LIN {X 0,Y 409.933,Z 400.183,A -85,B 0,C 180,E1 -10526.068,E2 -10526.068} C_VEL
LIN {X 0,Y 409.928,Z 401.653,A -85,B 0,C 180,E1 -10527.052,E2 -10527.052} C_VEL
LIN {X 0,Y 409.968,Z 402.683,A -85,B 0,C 180,E1 -10528.035,E2 -10528.035} C_VEL
LIN {X 0,Y 409.937,Z 403.318,A -85,B 0,C 180,E1 -10529.018,E2 -10529.018} C_VEL
LIN {X 0,Y 409.927,Z 403.562,A -85,B 0,C 180,E1 -10530,E2 -10530} C_VEL
LIN {X 0,Y 409.937,Z 403.388,A -85,B 0,C 180,E1 -10530.982,E2 -10530.982} C_VEL
LIN {X 0,Y 409.968,Z 402.792,A -85,B 0,C 180,E1 -10531.965,E2 -10531.965} C_VEL
LIN {X 0,Y 409.933,Z 400.415,A -85,B 0,C 180,E1 -10533.932,E2 -10533.932} C_VEL
LIN {X 0,Y 410.02,Z 397.492,A -85,B 0,C 180,E1 -10535.409,E2 -10535.409} C_VEL
LIN {X 0,Y 410.169,Z 393.533,A -85,B 0,C 180,E1 -10536.888,E2 -10536.888} C_VEL
LIN {X 0,Y 410.424,Z 388.44,A -85,B 0,C 180,E1 -10538.369,E2 -10538.369} C_VEL
LIN {X 0,Y 410.834,Z 382.051,A -85,B 0,C 180,E1 -10539.849,E2 -10539.849} C_VEL
LIN {X 0,Y 411.43,Z 374.069,A -85,B 0,C 180,E1 -10541.329,E2 -10541.329} C_VEL
LIN {X 0,Y 412.303,Z 364.173,A -85,B 0,C 180,E1 -10542.802,E2 -10542.802} C_VEL
LIN {X 0,Y 412.887,Z 354.848,A -85,B 0,C 180,E1 -10543.93,E2 -10543.93} C_VEL
LIN {X 0,Y 413.712,Z 343.698,A -85,B 0,C 180,E1 -10545.014,E2 -10545.014} C_VEL
LIN {X 0,Y 414.567,Z 332.678,A -85,B 0,C 180,E1 -10545.864,E2 -10545.864} C_VEL
LIN {X 0,Y 414.903,Z 324.983,A -85,B 0,C 180,E1 -10546.356,E2 -10546.356} C_VEL
LIN {X 0,Y 413.288,Z 311.721,A -85,B 0,C 180,E1 -10547.105,E2 -10547.105} C_VEL
LIN {X 0,Y 410.881,Z 298.907,A -85,B 0,C 180,E1 -10547.674,E2 -10547.674} C_VEL
LIN {X 0,Y 410.406,Z 296.498,A -85,B 0,C 180,E1 -10547.759,E2 -10547.759} C_VEL
LIN {X 0,Y 410.712,Z 289.615,A -85,B 0,C 180,E1 -10551.059,E2 -10551.059} C_VEL
LIN {X 0,Y 410.994,Z 283.191,A -85,B 0,C 180,E1 -10554.229,E2 -10554.229} C_VEL
LIN {X 0,Y 411.373,Z 276.838,A -85,B 0,C 180,E1 -10557.469,E2 -10557.469} C_VEL
LIN {X 0,Y 411.844,Z 270.571,A -85,B 0,C 180,E1 -10560.792,E2 -10560.792} C_VEL
LIN {X 0,Y 412.452,Z 264.434,A -85,B 0,C 180,E1 -10564.214,E2 -10564.214} C_VEL
LIN {X 0,Y 412.379,Z 260.162,A -85,B 0,C 180,E1 -10566.773,E2 -10566.773} C_VEL
LIN {X 0,Y 411.758,Z 255.497,A -85,B 0,C 180,E1 -10569.818,E2 -10569.818} C_VEL
LIN {X 0,Y 411.207,Z 252.267,A -85,B 0,C 180,E1 -10572.13,E2 -10572.13} C_VEL
LIN {X 0,Y 411.176,Z 252.27,A -85,B 0,C 180,E1 -10575.509,E2 -10575.509} C_VEL
LIN {X 0,Y 411.199,Z 252.27,A -85,B 0,C 180,E1 -10578.765,E2 -10578.765} C_VEL
LIN {X 0,Y 411.203,Z 252.267,A -85,B 0,C 180,E1 -10582.026,E2 -10582.026} C_VEL
LIN {X 0,Y 411.204,Z 252.266,A -85,B 0,C 180,E1 -10585.665,E2 -10585.665} C_VEL
LIN {X 0,Y 411.195,Z 252.267,A -85,B 0,C 180,E1 -10589.152,E2 -10589.152} C_VEL
LIN {X 0,Y 411.256,Z 252.258,A -85,B 0,C 180,E1 -10592.521,E2 -10592.521} C_VEL
LIN {X 0,Y 411.223,Z 252.264,A -85,B 0,C 180,E1 -10595.783,E2 -10595.783} C_VEL
LIN {X 0,Y 411.191,Z 252.267,A -85,B 0,C 180,E1 -10598.965,E2 -10598.965} C_VEL
LIN {X 0,Y 411.247,Z 252.262,A -85,B 0,C 180,E1 -10602.084,E2 -10602.084} C_VEL
LIN {X 0,Y 411.254,Z 252.26,A -85,B 0,C 180,E1 -10605.146,E2 -10605.146} C_VEL
LIN {X 0,Y 411.279,Z 252.257,A -85,B 0,C 180,E1 -10608.166,E2 -10608.166} C_VEL
LIN {X 0,Y 411.475,Z 252.232,A -85,B 0,C 180,E1 -10612.145,E2 -10612.145} C_VEL
LIN {X 0,Y 411.468,Z 252.233,A -85,B 0,C 180,E1 -10614.117,E2 -10614.117} C_VEL
LIN {X 0,Y 411.506,Z 252.228,A -85,B 0,C 180,E1 -10618.041,E2 -10618.041} C_VEL
LIN {X 0,Y 411.634,Z 252.212,A -85,B 0,C 180,E1 -10619.999,E2 -10619.999} C_VEL
LIN {X 0,Y 411.46,Z 252.236,A -85,B 0,C 180,E1 -10622.936,E2 -10622.936} C_VEL
LIN {X 0,Y 411.452,Z 252.236,A -85,B 0,C 180,E1 -10626.866,E2 -10626.866} C_VEL
LIN {X 0,Y 411.354,Z 252.446,A -85,B 0,C 180,E1 -10628.844,E2 -10628.844} C_VEL
LIN {X 0,Y 411.368,Z 255.81,A -85,B 0,C 180,E1 -10631.829,E2 -10631.829} C_VEL
LIN {X 0,Y 411.223,Z 258.159,A -85,B 0,C 180,E1 -10633.842,E2 -10633.842} C_VEL
LIN {X 0,Y 411.047,Z 261.892,A -85,B 0,C 180,E1 -10636.896,E2 -10636.896} C_VEL
LIN {X 0,Y 410.791,Z 265.812,A -85,B 0,C 180,E1 -10640.008,E2 -10640.008} C_VEL
LIN {X 0,Y 410.58,Z 269.911,A -85,B 0,C 180,E1 -10643.183,E2 -10643.183} C_VEL
LIN {X 0,Y 410.391,Z 274.236,A -85,B 0,C 180,E1 -10646.438,E2 -10646.438} C_VEL
LIN {X 0,Y 410.331,Z 276.757,A -85,B 0,C 180,E1 -10648.307,E2 -10648.307} C_VEL
LIN {X 0,Y 414.045,Z 291.96,A -85,B 0,C 180,E1 -10649.053,E2 -10649.053} C_VEL
LIN {X 0,Y 415.423,Z 299.541,A -85,B 0,C 180,E1 -10649.501,E2 -10649.501} C_VEL
LIN {X 0,Y 414.931,Z 311.573,A -85,B 0,C 180,E1 -10650.253,E2 -10650.253} C_VEL
LIN {X 0,Y 414.2,Z 322.984,A -85,B 0,C 180,E1 -10651.164,E2 -10651.164} C_VEL
LIN {X 0,Y 413.404,Z 333.611,A -85,B 0,C 180,E1 -10652.232,E2 -10652.232} C_VEL
LIN {X 0,Y 412.54,Z 344.203,A -85,B 0,C 180,E1 -10653.568,E2 -10653.568} C_VEL
LIN {X 0,Y 411.775,Z 353.273,A -85,B 0,C 180,E1 -10654.993,E2 -10654.993} C_VEL
LIN {X 0,Y 411.141,Z 361.113,A -85,B 0,C 180,E1 -10656.545,E2 -10656.545} C_VEL
LIN {X 0,Y 410.667,Z 367.275,A -85,B 0,C 180,E1 -10658.075,E2 -10658.075} C_VEL
LIN {X 0,Y 410.326,Z 372.035,A -85,B 0,C 180,E1 -10659.58,E2 -10659.58} C_VEL
LIN {X 0,Y 410.099,Z 375.597,A -85,B 0,C 180,E1 -10661.06,E2 -10661.06} C_VEL
LIN {X 0,Y 409.93,Z 378.103,A -85,B 0,C 180,E1 -10662.507,E2 -10662.507} C_VEL
LIN {X 0,Y 409.84,Z 379.686,A -85,B 0,C 180,E1 -10663.929,E2 -10663.929} C_VEL
LIN {X 0,Y 409.775,Z 380.432,A -85,B 0,C 180,E1 -10665.318,E2 -10665.318} C_VEL
LIN {X 0,Y 409.739,Z 380.392,A -85,B 0,C 180,E1 -10666.679,E2 -10666.679} C_VEL
LIN {X 0,Y 409.781,Z 379.571,A -85,B 0,C 180,E1 -10668.021,E2 -10668.021} C_VEL
LIN {X 0,Y 409.877,Z 378.049,A -85,B 0,C 180,E1 -10669.341,E2 -10669.341} C_VEL
LIN {X 0,Y 410.003,Z 375.839,A -85,B 0,C 180,E1 -10670.638,E2 -10670.638} C_VEL
LIN {X 0,Y 410.322,Z 370.969,A -85,B 0,C 180,E1 -10672.595,E2 -10672.595} C_VEL
LIN {X 0,Y 410.649,Z 366.267,A -85,B 0,C 180,E1 -10674.002,E2 -10674.002} C_VEL
LIN {X 0,Y 411.05,Z 359.297,A -85,B 0,C 180,E1 -10675.653,E2 -10675.653} C_VEL
LIN {X 0,Y 411.696,Z 351.038,A -85,B 0,C 180,E1 -10677.181,E2 -10677.181} C_VEL
LIN {X 0,Y 412.311,Z 342.559,A -85,B 0,C 180,E1 -10678.456,E2 -10678.456} C_VEL
LIN {X 0,Y 412.941,Z 333,A -85,B 0,C 180,E1 -10679.636,E2 -10679.636} C_VEL
LIN {X 0,Y 413.603,Z 323.215,A -85,B 0,C 180,E1 -10680.618,E2 -10680.618} C_VEL
LIN {X 0,Y 414.317,Z 311.202,A -85,B 0,C 180,E1 -10681.575,E2 -10681.575} C_VEL
LIN {X 0,Y 414.99,Z 300.07,A -85,B 0,C 180,E1 -10682.261,E2 -10682.261} C_VEL
LIN {X 0,Y 412.651,Z 287.184,A -85,B 0,C 180,E1 -10682.965,E2 -10682.965} C_VEL
LIN {X 0,Y 410.191,Z 276.058,A -85,B 0,C 180,E1 -10683.425,E2 -10683.425} C_VEL
LIN {X 0,Y 410.335,Z 271.318,A -85,B 0,C 180,E1 -10686.801,E2 -10686.801} C_VEL
LIN {X 0,Y 410.554,Z 266.488,A -85,B 0,C 180,E1 -10690.302,E2 -10690.302} C_VEL
LIN {X 0,Y 410.726,Z 262.34,A -85,B 0,C 180,E1 -10693.374,E2 -10693.374} C_VEL
LIN {X 0,Y 410.976,Z 257.338,A -85,B 0,C 180,E1 -10697.156,E2 -10697.156} C_VEL
LIN {X 0,Y 411.091,Z 253.482,A -85,B 0,C 180,E1 -10700.157,E2 -10700.157} C_VEL
LIN {X 0,Y 411.12,Z 252.276,A -85,B 0,C 180,E1 -10701.15,E2 -10701.15} C_VEL
LIN {X 0,Y 411.404,Z 252.241,A -85,B 0,C 180,E1 -10703.132,E2 -10703.132} C_VEL
LIN {X 0,Y 411.301,Z 252.252,A -85,B 0,C 180,E1 -10705.099,E2 -10705.099} C_VEL
LIN {X 0,Y 411.481,Z 252.228,A -85,B 0,C 180,E1 -10708.307,E2 -10708.307} C_VEL
LIN {X 0,Y 411.633,Z 252.211,A -85,B 0,C 180,E1 -10710,E2 -10710} C_VEL
LIN {X 0,Y 411.46,Z 252.231,A -85,B 0,C 180,E1 -10712.571,E2 -10712.571} C_VEL
LIN {X 0,Y 410.775,Z 252.318,A -85,B 0,C 180,E1 -10713.387,E2 -10713.387} C_VEL
LIN {X 0,Y 407.897,Z 252.677,A -85,B 0,C 180,E1 -10714.712,E2 -10714.712} C_VEL
LIN {X 0,Y 405.484,Z 252.976,A -85,B 0,C 180,E1 -10715.783,E2 -10715.783} C_VEL
LIN {X 0,Y 404.469,Z 253.105,A -85,B 0,C 180,E1 -10716.611,E2 -10716.611} C_VEL
LIN {X 0,Y 404.397,Z 253.11,A -85,B 0,C 180,E1 -10716.891,E2 -10716.891} C_VEL
LIN {X 0,Y 404.286,Z 253.125,A -85,B 0,C 180,E1 -10719.001,E2 -10719.001} C_VEL
LIN {X 0,Y 404.26,Z 253.131,A -85,B 0,C 180,E1 -10722.041,E2 -10722.041} C_VEL
LIN {X 0,Y 404.202,Z 253.135,A -85,B 0,C 180,E1 -10725.118,E2 -10725.118} C_VEL
LIN {X 0,Y 404.203,Z 253.138,A -85,B 0,C 180,E1 -10728.238,E2 -10728.238} C_VEL
LIN {X 0,Y 404.169,Z 253.14,A -85,B 0,C 180,E1 -10731.417,E2 -10731.417} C_VEL
LIN {X 0,Y 404.167,Z 253.14,A -85,B 0,C 180,E1 -10734.666,E2 -10734.666} C_VEL
LIN {X 0,Y 404.187,Z 253.14,A -85,B 0,C 180,E1 -10738,E2 -10738} C_VEL
LIN {X 0,Y 404.135,Z 253.146,A -85,B 0,C 180,E1 -10741.56,E2 -10741.56} C_VEL
LIN {X 0,Y 404.174,Z 253.139,A -85,B 0,C 180,E1 -10745.017,E2 -10745.017} C_VEL
LIN {X 0,Y 404.153,Z 253.14,A -85,B 0,C 180,E1 -10748.756,E2 -10748.756} C_VEL
LIN {X 0,Y 404.181,Z 253.141,A -85,B 0,C 180,E1 -10751.611,E2 -10751.611} C_VEL
LIN {X 0,Y 404.19,Z 253.136,A -85,B 0,C 180,E1 -10754.531,E2 -10754.531} C_VEL
LIN {X 0,Y 404.196,Z 253.139,A -85,B 0,C 180,E1 -10757.306,E2 -10757.306} C_VEL
LIN {X 0,Y 404.158,Z 253.141,A -85,B 0,C 180,E1 -10759.956,E2 -10759.956} C_VEL
LIN {X 0,Y 404.131,Z 253.147,A -85,B 0,C 180,E1 -10763.125,E2 -10763.125} C_VEL
LIN {X 0,Y 404.135,Z 253.143,A -85,B 0,C 180,E1 -10766.189,E2 -10766.189} C_VEL
LIN {X 0,Y 404.144,Z 253.142,A -85,B 0,C 180,E1 -10769.716,E2 -10769.716} C_VEL
LIN {X 0,Y 404.186,Z 253.14,A -85,B 0,C 180,E1 -10773.124,E2 -10773.124} C_VEL
LIN {X 0,Y 404.168,Z 253.141,A -85,B 0,C 180,E1 -10775.335,E2 -10775.335} C_VEL
LIN {X 0,Y 404.13,Z 253.147,A -85,B 0,C 180,E1 -10778.582,E2 -10778.582} C_VEL
LIN {X 0,Y 404.202,Z 253.135,A -85,B 0,C 180,E1 -10781.763,E2 -10781.763} C_VEL
LIN {X 0,Y 404.198,Z 253.139,A -85,B 0,C 180,E1 -10784.883,E2 -10784.883} C_VEL
LIN {X 0,Y 404.249,Z 253.13,A -85,B 0,C 180,E1 -10787.96,E2 -10787.96} C_VEL
LIN {X 0,Y 404.398,Z 253.113,A -85,B 0,C 180,E1 -10792.13,E2 -10792.13} C_VEL
LIN {X 0,Y 404.416,Z 253.111,A -85,B 0,C 180,E1 -10794.016,E2 -10794.016} C_VEL
LIN {X 0,Y 404.476,Z 253.103,A -85,B 0,C 180,E1 -10798.01,E2 -10798.01} C_VEL
LIN {X 0,Y 404.605,Z 253.088,A -85,B 0,C 180,E1 -10800.001,E2 -10800.001} C_VEL
LIN {X 0,Y 404.418,Z 253.108,A -85,B 0,C 180,E1 -10802.99,E2 -10802.99} C_VEL
LIN {X 0,Y 404.406,Z 253.109,A -85,B 0,C 180,E1 -10806.988,E2 -10806.988} C_VEL
LIN {X 0,Y 404.266,Z 253.13,A -85,B 0,C 180,E1 -10810.013,E2 -10810.013} C_VEL
LIN {X 0,Y 404.263,Z 253.128,A -85,B 0,C 180,E1 -10813.213,E2 -10813.213} C_VEL
LIN {X 0,Y 404.212,Z 253.133,A -85,B 0,C 180,E1 -10817.008,E2 -10817.008} C_VEL
LIN {X 0,Y 404.161,Z 253.14,A -85,B 0,C 180,E1 -10820.353,E2 -10820.353} C_VEL
LIN {X 0,Y 404.167,Z 253.143,A -85,B 0,C 180,E1 -10823.576,E2 -10823.576} C_VEL
LIN {X 0,Y 404.182,Z 253.141,A -85,B 0,C 180,E1 -10825.768,E2 -10825.768} C_VEL
LIN {X 0,Y 404.193,Z 253.138,A -85,B 0,C 180,E1 -10828.001,E2 -10828.001} C_VEL
LIN {X 0,Y 404.138,Z 253.146,A -85,B 0,C 180,E1 -10831.559,E2 -10831.559} C_VEL
LIN {X 0,Y 404.184,Z 253.14,A -85,B 0,C 180,E1 -10835.017,E2 -10835.017} C_VEL
LIN {X 0,Y 404.157,Z 253.142,A -85,B 0,C 180,E1 -10838.758,E2 -10838.758} C_VEL
LIN {X 0,Y 404.123,Z 253.146,A -85,B 0,C 180,E1 -10841.601,E2 -10841.601} C_VEL
LIN {X 0,Y 404.146,Z 253.143,A -85,B 0,C 180,E1 -10844.523,E2 -10844.523} C_VEL
LIN {X 0,Y 404.137,Z 253.147,A -85,B 0,C 180,E1 -10847.297,E2 -10847.297} C_VEL
LIN {X 0,Y 404.193,Z 253.241,A -85,B 0,C 180,E1 -10849.222,E2 -10849.222} C_VEL
LIN {X 0,Y 405.002,Z 257.819,A -85,B 0,C 180,E1 -10852.003,E2 -10852.003} C_VEL
LIN {X 0,Y 405.39,Z 262.275,A -85,B 0,C 180,E1 -10854.57,E2 -10854.57} C_VEL
LIN {X 0,Y 405.055,Z 267.592,A -85,B 0,C 180,E1 -10857.462,E2 -10857.462} C_VEL
LIN {X 0,Y 404.493,Z 274.108,A -85,B 0,C 180,E1 -10860.89,E2 -10860.89} C_VEL
LIN {X 0,Y 404.056,Z 281.663,A -85,B 0,C 180,E1 -10864.753,E2 -10864.753} C_VEL
LIN {X 0,Y 403.719,Z 288.235,A -85,B 0,C 180,E1 -10868.021,E2 -10868.021} C_VEL
LIN {X 0,Y 403.451,Z 294.748,A -85,B 0,C 180,E1 -10871.2,E2 -10871.2} C_VEL
LIN {X 0,Y 403.357,Z 297.222,A -85,B 0,C 180,E1 -10872.308,E2 -10872.308} C_VEL
LIN {X 0,Y 405.673,Z 310.351,A -85,B 0,C 180,E1 -10872.827,E2 -10872.827} C_VEL
LIN {X 0,Y 407.456,Z 323.993,A -85,B 0,C 180,E1 -10873.57,E2 -10873.57} C_VEL
LIN {X 0,Y 407.412,Z 330.524,A -85,B 0,C 180,E1 -10873.978,E2 -10873.978} C_VEL
LIN {X 0,Y 406.585,Z 342.104,A -85,B 0,C 180,E1 -10874.844,E2 -10874.844} C_VEL
LIN {X 0,Y 405.723,Z 353.789,A -85,B 0,C 180,E1 -10875.965,E2 -10875.965} C_VEL
LIN {X 0,Y 405.064,Z 364.197,A -85,B 0,C 180,E1 -10877.22,E2 -10877.22} C_VEL
LIN {X 0,Y 404.208,Z 374.12,A -85,B 0,C 180,E1 -10878.72,E2 -10878.72} C_VEL
LIN {X 0,Y 403.675,Z 382.113,A -85,B 0,C 180,E1 -10880.227,E2 -10880.227} C_VEL
LIN {X 0,Y 403.366,Z 387.519,A -85,B 0,C 180,E1 -10881.483,E2 -10881.483} C_VEL
LIN {X 0,Y 403.082,Z 392.807,A -85,B 0,C 180,E1 -10882.99,E2 -10882.99} C_VEL
LIN {X 0,Y 402.918,Z 396.908,A -85,B 0,C 180,E1 -10884.495,E2 -10884.495} C_VEL
LIN {X 0,Y 402.854,Z 399.941,A -85,B 0,C 180,E1 -10885.998,E2 -10885.998} C_VEL
LIN {X 0,Y 402.827,Z 401.426,A -85,B 0,C 180,E1 -10887,E2 -10887} C_VEL
LIN {X 0,Y 402.866,Z 402.464,A -85,B 0,C 180,E1 -10888,E2 -10888} C_VEL
LIN {X 0,Y 402.864,Z 403.106,A -85,B 0,C 180,E1 -10889,E2 -10889} C_VEL
LIN {X 0,Y 402.852,Z 403.358,A -85,B 0,C 180,E1 -10890,E2 -10890} C_VEL
LIN {X 0,Y 402.864,Z 403.199,A -85,B 0,C 180,E1 -10890.999,E2 -10890.999} C_VEL
LIN {X 0,Y 402.866,Z 402.609,A -85,B 0,C 180,E1 -10891.999,E2 -10891.999} C_VEL
LIN {X 0,Y 402.853,Z 400.245,A -85,B 0,C 180,E1 -10894.001,E2 -10894.001} C_VEL
LIN {X 0,Y 402.918,Z 397.334,A -85,B 0,C 180,E1 -10895.505,E2 -10895.505} C_VEL
LIN {X 0,Y 403.082,Z 393.389,A -85,B 0,C 180,E1 -10897.01,E2 -10897.01} C_VEL
LIN {X 0,Y 403.366,Z 388.31,A -85,B 0,C 180,E1 -10898.516,E2 -10898.516} C_VEL
LIN {X 0,Y 403.824,Z 381.942,A -85,B 0,C 180,E1 -10900.022,E2 -10900.022} C_VEL
LIN {X 0,Y 404.429,Z 373.983,A -85,B 0,C 180,E1 -10901.527,E2 -10901.527} C_VEL
LIN {X 0,Y 405.353,Z 364.109,A -85,B 0,C 180,E1 -10903.026,E2 -10903.026} C_VEL
LIN {X 0,Y 406.022,Z 354.346,A -85,B 0,C 180,E1 -10904.225,E2 -10904.225} C_VEL
LIN {X 0,Y 406.861,Z 343.762,A -85,B 0,C 180,E1 -10905.273,E2 -10905.273} C_VEL
LIN {X 0,Y 407.75,Z 332.866,A -85,B 0,C 180,E1 -10906.134,E2 -10906.134} C_VEL
LIN {X 0,Y 408.015,Z 325.458,A -85,B 0,C 180,E1 -10906.628,E2 -10906.628} C_VEL
LIN {X 0,Y 406.532,Z 312.758,A -85,B 0,C 180,E1 -10907.375,E2 -10907.375} C_VEL
LIN {X 0,Y 404.064,Z 299.804,A -85,B 0,C 180,E1 -10907.982,E2 -10907.982} C_VEL
LIN {X 0,Y 403.377,Z 296.306,A -85,B 0,C 180,E1 -10908.112,E2 -10908.112} C_VEL
LIN {X 0,Y 403.662,Z 289.507,A -85,B 0,C 180,E1 -10911.445,E2 -10911.445} C_VEL
LIN {X 0,Y 404.001,Z 283.107,A -85,B 0,C 180,E1 -10914.676,E2 -10914.676} C_VEL
LIN {X 0,Y 404.388,Z 276.776,A -85,B 0,C 180,E1 -10917.984,E2 -10917.984} C_VEL
LIN {X 0,Y 405.008,Z 269.916,A -85,B 0,C 180,E1 -10921.756,E2 -10921.756} C_VEL
LIN {X 0,Y 405.468,Z 264.438,A -85,B 0,C 180,E1 -10924.888,E2 -10924.888} C_VEL
LIN {X 0,Y 405.286,Z 260.478,A -85,B 0,C 180,E1 -10927.367,E2 -10927.367} C_VEL
LIN {X 0,Y 404.687,Z 256.34,A -85,B 0,C 180,E1 -10930.17,E2 -10930.17} C_VEL
LIN {X 0,Y 404.159,Z 253.144,A -85,B 0,C 180,E1 -10932.557,E2 -10932.557} C_VEL
LIN {X 0,Y 404.148,Z 253.147,A -85,B 0,C 180,E1 -10935.925,E2 -10935.925} C_VEL
LIN {X 0,Y 404.151,Z 253.147,A -85,B 0,C 180,E1 -10938.638,E2 -10938.638} C_VEL
LIN {X 0,Y 404.16,Z 253.145,A -85,B 0,C 180,E1 -10941.489,E2 -10941.489} C_VEL
LIN {X 0,Y 404.183,Z 253.14,A -85,B 0,C 180,E1 -10944.983,E2 -10944.983} C_VEL
LIN {X 0,Y 404.143,Z 253.145,A -85,B 0,C 180,E1 -10948.553,E2 -10948.553} C_VEL
LIN {X 0,Y 404.194,Z 253.138,A -85,B 0,C 180,E1 -10951.999,E2 -10951.999} C_VEL
LIN {X 0,Y 404.173,Z 253.141,A -85,B 0,C 180,E1 -10955.333,E2 -10955.333} C_VEL
LIN {X 0,Y 404.134,Z 253.146,A -85,B 0,C 180,E1 -10958.579,E2 -10958.579} C_VEL
LIN {X 0,Y 404.205,Z 253.137,A -85,B 0,C 180,E1 -10961.761,E2 -10961.761} C_VEL
LIN {X 0,Y 404.2,Z 253.138,A -85,B 0,C 180,E1 -10964.881,E2 -10964.881} C_VEL
LIN {X 0,Y 404.251,Z 253.131,A -85,B 0,C 180,E1 -10967.957,E2 -10967.957} C_VEL
LIN {X 0,Y 404.427,Z 253.11,A -85,B 0,C 180,E1 -10972.098,E2 -10972.098} C_VEL
LIN {X 0,Y 404.417,Z 253.111,A -85,B 0,C 180,E1 -10974.014,E2 -10974.014} C_VEL
LIN {X 0,Y 404.475,Z 253.104,A -85,B 0,C 180,E1 -10978.007,E2 -10978.007} C_VEL
LIN {X 0,Y 404.603,Z 253.088,A -85,B 0,C 180,E1 -10979.999,E2 -10979.999} C_VEL
LIN {X 0,Y 404.417,Z 253.114,A -85,B 0,C 180,E1 -10982.987,E2 -10982.987} C_VEL
LIN {X 0,Y 404.398,Z 253.115,A -85,B 0,C 180,E1 -10986.986,E2 -10986.986} C_VEL
LIN {X 0,Y 404.376,Z 253.118,A -85,B 0,C 180,E1 -10987.991,E2 -10987.991} C_VEL
LIN {X 0,Y 404.365,Z 253.737,A -85,B 0,C 180,E1 -10988.998,E2 -10988.998} C_VEL
LIN {X 0,Y 404.334,Z 257.099,A -85,B 0,C 180,E1 -10992.038,E2 -10992.038} C_VEL
LIN {X 0,Y 404.097,Z 260.696,A -85,B 0,C 180,E1 -10995.121,E2 -10995.121} C_VEL
LIN {X 0,Y 403.875,Z 264.511,A -85,B 0,C 180,E1 -10998.252,E2 -10998.252} C_VEL
LIN {X 0,Y 403.632,Z 268.511,A -85,B 0,C 180,E1 -11001.446,E2 -11001.446} C_VEL
LIN {X 0,Y 403.429,Z 273.172,A -85,B 0,C 180,E1 -11005.062,E2 -11005.062} C_VEL
LIN {X 0,Y 403.272,Z 276.979,A -85,B 0,C 180,E1 -11007.947,E2 -11007.947} C_VEL
LIN {X 0,Y 406.97,Z 291.921,A -85,B 0,C 180,E1 -11008.703,E2 -11008.703} C_VEL
LIN {X 0,Y 408.755,Z 302.254,A -85,B 0,C 180,E1 -11009.34,E2 -11009.34} C_VEL
LIN {X 0,Y 408.087,Z 313.529,A -85,B 0,C 180,E1 -11010.081,E2 -11010.081} C_VEL
LIN {X 0,Y 407.324,Z 324.098,A -85,B 0,C 180,E1 -11010.963,E2 -11010.963} C_VEL
LIN {X 0,Y 406.464,Z 334.838,A -85,B 0,C 180,E1 -11012.089,E2 -11012.089} C_VEL
LIN {X 0,Y 405.606,Z 344.714,A -85,B 0,C 180,E1 -11013.372,E2 -11013.372} C_VEL
LIN {X 0,Y 404.89,Z 352.697,A -85,B 0,C 180,E1 -11014.642,E2 -11014.642} C_VEL
LIN {X 0,Y 404.27,Z 359.623,A -85,B 0,C 180,E1 -11015.978,E2 -11015.978} C_VEL
LIN {X 0,Y 403.743,Z 366.123,A -85,B 0,C 180,E1 -11017.533,E2 -11017.533} C_VEL
LIN {X 0,Y 403.29,Z 372.051,A -85,B 0,C 180,E1 -11019.377,E2 -11019.377} C_VEL
LIN {X 0,Y 403.047,Z 375.464,A -85,B 0,C 180,E1 -11020.788,E2 -11020.788} C_VEL
LIN {X 0,Y 402.862,Z 377.979,A -85,B 0,C 180,E1 -11022.192,E2 -11022.192} C_VEL
LIN {X 0,Y 402.824,Z 378.914,A -85,B 0,C 180,E1 -11022.883,E2 -11022.883} C_VEL
LIN {X 0,Y 402.731,Z 380.235,A -85,B 0,C 180,E1 -11024.318,E2 -11024.318} C_VEL
LIN {X 0,Y 402.678,Z 380.697,A -85,B 0,C 180,E1 -11025.725,E2 -11025.725} C_VEL
LIN {X 0,Y 402.65,Z 380.375,A -85,B 0,C 180,E1 -11027.143,E2 -11027.143} C_VEL
LIN {X 0,Y 402.732,Z 379.19,A -85,B 0,C 180,E1 -11028.621,E2 -11028.621} C_VEL
LIN {X 0,Y 402.833,Z 377.042,A -85,B 0,C 180,E1 -11030.14,E2 -11030.14} C_VEL
LIN {X 0,Y 403.081,Z 373.838,A -85,B 0,C 180,E1 -11031.682,E2 -11031.682} C_VEL
LIN {X 0,Y 403.383,Z 369.38,A -85,B 0,C 180,E1 -11033.265,E2 -11033.265} C_VEL
LIN {X 0,Y 403.786,Z 363.222,A -85,B 0,C 180,E1 -11034.945,E2 -11034.945} C_VEL
LIN {X 0,Y 404.342,Z 355.751,A -85,B 0,C 180,E1 -11036.54,E2 -11036.54} C_VEL
LIN {X 0,Y 405.05,Z 346.647,A -85,B 0,C 180,E1 -11038.08,E2 -11038.08} C_VEL
LIN {X 0,Y 405.736,Z 336.849,A -85,B 0,C 180,E1 -11039.415,E2 -11039.415} C_VEL
LIN {X 0,Y 406.522,Z 325.674,A -85,B 0,C 180,E1 -11040.624,E2 -11040.624} C_VEL
LIN {X 0,Y 407.287,Z 313.794,A -85,B 0,C 180,E1 -11041.643,E2 -11041.643} C_VEL
LIN {X 0,Y 407.973,Z 302.84,A -85,B 0,C 180,E1 -11042.37,E2 -11042.37} C_VEL
LIN {X 0,Y 407.917,Z 299.95,A -85,B 0,C 180,E1 -11042.539,E2 -11042.539} C_VEL
LIN {X 0,Y 405.529,Z 287.07,A -85,B 0,C 180,E1 -11043.254,E2 -11043.254} C_VEL
LIN {X 0,Y 403.138,Z 276.246,A -85,B 0,C 180,E1 -11043.711,E2 -11043.711} C_VEL
LIN {X 0,Y 403.223,Z 272.558,A -85,B 0,C 180,E1 -11046.367,E2 -11046.367} C_VEL
LIN {X 0,Y 403.455,Z 268.129,A -85,B 0,C 180,E1 -11049.612,E2 -11049.612} C_VEL
LIN {X 0,Y 403.659,Z 263.268,A -85,B 0,C 180,E1 -11053.248,E2 -11053.248} C_VEL
LIN {X 0,Y 403.894,Z 258.357,A -85,B 0,C 180,E1 -11057.009,E2 -11057.009} C_VEL
LIN {X 0,Y 404.034,Z 254.575,A -85,B 0,C 180,E1 -11059.983,E2 -11059.983} C_VEL
LIN {X 0,Y 404.074,Z 253.314,A -85,B 0,C 180,E1 -11060.994,E2 -11060.994} C_VEL
LIN {X 0,Y 404.341,Z 253.12,A -85,B 0,C 180,E1 -11063.012,E2 -11063.012} C_VEL
LIN {X 0,Y 404.272,Z 253.128,A -85,B 0,C 180,E1 -11065.014,E2 -11065.014} C_VEL
LIN {X 0,Y 404.473,Z 253.102,A -85,B 0,C 180,E1 -11068.009,E2 -11068.009} C_VEL
LIN {X 0,Y 404.602,Z 253.087,A -85,B 0,C 180,E1 -11070,E2 -11070} C_VEL
LIN {X 0,Y 404.414,Z 253.11,A -85,B 0,C 180,E1 -11072.989,E2 -11072.989} C_VEL
LIN {X 0,Y 404.397,Z 253.11,A -85,B 0,C 180,E1 -11076.891,E2 -11076.891} C_VEL
LIN {X 0,Y 403.746,Z 253.194,A -85,B 0,C 180,E1 -11077.722,E2 -11077.722} C_VEL
LIN {X 0,Y 400.847,Z 253.557,A -85,B 0,C 180,E1 -11079.069,E2 -11079.069} C_VEL
LIN {X 0,Y 398.367,Z 253.865,A -85,B 0,C 180,E1 -11080.158,E2 -11080.158} C_VEL
LIN {X 0,Y 397.29,Z 253.996,A -85,B 0,C 180,E1 -11081.001,E2 -11081.001} C_VEL
LIN {X 0,Y 397.197,Z 254.007,A -85,B 0,C 180,E1 -11081.287,E2 -11081.287} C_VEL
LIN {X 0,Y 397.172,Z 254.014,A -85,B 0,C 180,E1 -11084.343,E2 -11084.343} C_VEL
LIN {X 0,Y 397.165,Z 254.012,A -85,B 0,C 180,E1 -11087.507,E2 -11087.507} C_VEL
LIN {X 0,Y 397.122,Z 254.017,A -85,B 0,C 180,E1 -11090.729,E2 -11090.729} C_VEL
LIN {X 0,Y 397.124,Z 254.02,A -85,B 0,C 180,E1 -11094.018,E2 -11094.018} C_VEL
LIN {X 0,Y 397.184,Z 254.011,A -85,B 0,C 180,E1 -11097.39,E2 -11097.39} C_VEL
LIN {X 0,Y 397.075,Z 254.023,A -85,B 0,C 180,E1 -11100.882,E2 -11100.882} C_VEL
LIN {X 0,Y 397.115,Z 254.018,A -85,B 0,C 180,E1 -11104.494,E2 -11104.494} C_VEL
LIN {X 0,Y 397.099,Z 254.019,A -85,B 0,C 180,E1 -11108.275,E2 -11108.275} C_VEL
LIN {X 0,Y 397.146,Z 254.015,A -85,B 0,C 180,E1 -11111.994,E2 -11111.994} C_VEL
LIN {X 0,Y 397.14,Z 254.017,A -85,B 0,C 180,E1 -11115.06,E2 -11115.06} C_VEL
LIN {X 0,Y 397.145,Z 254.014,A -85,B 0,C 180,E1 -11118.008,E2 -11118.008} C_VEL
LIN {X 0,Y 397.1,Z 254.021,A -85,B 0,C 180,E1 -11121.727,E2 -11121.727} C_VEL
LIN {X 0,Y 397.116,Z 254.02,A -85,B 0,C 180,E1 -11125.508,E2 -11125.508} C_VEL
LIN {X 0,Y 397.075,Z 254.026,A -85,B 0,C 180,E1 -11129.119,E2 -11129.119} C_VEL
LIN {X 0,Y 397.186,Z 254.012,A -85,B 0,C 180,E1 -11132.611,E2 -11132.611} C_VEL
LIN {X 0,Y 397.124,Z 254.016,A -85,B 0,C 180,E1 -11135.983,E2 -11135.983} C_VEL
LIN {X 0,Y 397.13,Z 254.015,A -85,B 0,C 180,E1 -11139.706,E2 -11139.706} C_VEL
LIN {X 0,Y 397.174,Z 254.014,A -85,B 0,C 180,E1 -11142.846,E2 -11142.846} C_VEL
LIN {X 0,Y 397.221,Z 254.008,A -85,B 0,C 180,E1 -11146.704,E2 -11146.704} C_VEL
LIN {X 0,Y 397.211,Z 254.005,A -85,B 0,C 180,E1 -11149.81,E2 -11149.81} C_VEL
LIN {X 0,Y 397.346,Z 253.991,A -85,B 0,C 180,E1 -11152.889,E2 -11152.889} C_VEL
LIN {X 0,Y 397.248,Z 254.002,A -85,B 0,C 180,E1 -11154.926,E2 -11154.926} C_VEL
LIN {X 0,Y 397.445,Z 253.979,A -85,B 0,C 180,E1 -11157.974,E2 -11157.974} C_VEL
LIN {X 0,Y 397.574,Z 253.964,A -85,B 0,C 180,E1 -11160.001,E2 -11160.001} C_VEL
LIN {X 0,Y 397.376,Z 253.985,A -85,B 0,C 180,E1 -11163.043,E2 -11163.043} C_VEL
LIN {X 0,Y 397.359,Z 253.987,A -85,B 0,C 180,E1 -11167.113,E2 -11167.113} C_VEL
LIN {X 0,Y 397.224,Z 254.008,A -85,B 0,C 180,E1 -11170.192,E2 -11170.192} C_VEL
LIN {X 0,Y 397.223,Z 254.005,A -85,B 0,C 180,E1 -11173.322,E2 -11173.322} C_VEL
LIN {X 0,Y 397.179,Z 254.01,A -85,B 0,C 180,E1 -11177.156,E2 -11177.156} C_VEL
LIN {X 0,Y 397.1,Z 254.019,A -85,B 0,C 180,E1 -11180.731,E2 -11180.731} C_VEL
LIN {X 0,Y 397.13,Z 254.018,A -85,B 0,C 180,E1 -11184.019,E2 -11184.019} C_VEL
LIN {X 0,Y 397.192,Z 254.012,A -85,B 0,C 180,E1 -11187.391,E2 -11187.391} C_VEL
LIN {X 0,Y 397.077,Z 254.023,A -85,B 0,C 180,E1 -11190.884,E2 -11190.884} C_VEL
LIN {X 0,Y 397.125,Z 254.016,A -85,B 0,C 180,E1 -11194.494,E2 -11194.494} C_VEL
LIN {X 0,Y 397.105,Z 254.019,A -85,B 0,C 180,E1 -11198.276,E2 -11198.276} C_VEL
LIN {X 0,Y 397.089,Z 254.024,A -85,B 0,C 180,E1 -11200.91,E2 -11200.91} C_VEL
LIN {X 0,Y 397.101,Z 254.021,A -85,B 0,C 180,E1 -11203.65,E2 -11203.65} C_VEL
LIN {X 0,Y 397.103,Z 254.023,A -85,B 0,C 180,E1 -11206.522,E2 -11206.522} C_VEL
LIN {X 0,Y 397.133,Z 254.122,A -85,B 0,C 180,E1 -11209.014,E2 -11209.014} C_VEL
LIN {X 0,Y 397.935,Z 258.663,A -85,B 0,C 180,E1 -11211.82,E2 -11211.82} C_VEL
LIN {X 0,Y 398.355,Z 263.028,A -85,B 0,C 180,E1 -11214.395,E2 -11214.395} C_VEL
LIN {X 0,Y 398.038,Z 268.469,A -85,B 0,C 180,E1 -11217.418,E2 -11217.418} C_VEL
LIN {X 0,Y 397.433,Z 274.993,A -85,B 0,C 180,E1 -11220.903,E2 -11220.903} C_VEL
LIN {X 0,Y 396.961,Z 282.583,A -85,B 0,C 180,E1 -11224.856,E2 -11224.856} C_VEL
LIN {X 0,Y 396.622,Z 289.091,A -85,B 0,C 180,E1 -11228.154,E2 -11228.154} C_VEL
LIN {X 0,Y 396.337,Z 295.59,A -85,B 0,C 180,E1 -11231.387,E2 -11231.387} C_VEL
LIN {X 0,Y 396.285,Z 296.809,A -85,B 0,C 180,E1 -11231.987,E2 -11231.987} C_VEL
LIN {X 0,Y 398.934,Z 312.219,A -85,B 0,C 180,E1 -11232.647,E2 -11232.647} C_VEL
LIN {X 0,Y 400.605,Z 325.587,A -85,B 0,C 180,E1 -11233.415,E2 -11233.415} C_VEL
LIN {X 0,Y 400.085,Z 336.925,A -85,B 0,C 180,E1 -11234.2,E2 -11234.2} C_VEL
LIN {X 0,Y 399.202,Z 348.433,A -85,B 0,C 180,E1 -11235.21,E2 -11235.21} C_VEL
LIN {X 0,Y 398.43,Z 358.574,A -85,B 0,C 180,E1 -11236.322,E2 -11236.322} C_VEL
LIN {X 0,Y 397.83,Z 367.374,A -85,B 0,C 180,E1 -11237.502,E2 -11237.502} C_VEL
LIN {X 0,Y 396.98,Z 376.617,A -85,B 0,C 180,E1 -11239.029,E2 -11239.029} C_VEL
LIN {X 0,Y 396.488,Z 384.054,A -85,B 0,C 180,E1 -11240.563,E2 -11240.563} C_VEL
LIN {X 0,Y 396.192,Z 389.107,A -85,B 0,C 180,E1 -11241.842,E2 -11241.842} C_VEL
LIN {X 0,Y 395.924,Z 394.003,A -85,B 0,C 180,E1 -11243.375,E2 -11243.375} C_VEL
LIN {X 0,Y 395.845,Z 397.761,A -85,B 0,C 180,E1 -11244.907,E2 -11244.907} C_VEL
LIN {X 0,Y 395.776,Z 399.694,A -85,B 0,C 180,E1 -11245.927,E2 -11245.927} C_VEL
LIN {X 0,Y 395.73,Z 401.195,A -85,B 0,C 180,E1 -11246.946,E2 -11246.946} C_VEL
LIN {X 0,Y 395.765,Z 402.243,A -85,B 0,C 180,E1 -11247.965,E2 -11247.965} C_VEL
LIN {X 0,Y 395.792,Z 402.894,A -85,B 0,C 180,E1 -11248.982,E2 -11248.982} C_VEL
LIN {X 0,Y 395.779,Z 403.153,A -85,B 0,C 180,E1 -11250,E2 -11250} C_VEL
LIN {X 0,Y 395.792,Z 403.008,A -85,B 0,C 180,E1 -11251.017,E2 -11251.017} C_VEL
LIN {X 0,Y 395.764,Z 402.426,A -85,B 0,C 180,E1 -11252.035,E2 -11252.035} C_VEL
LIN {X 0,Y 395.776,Z 400.075,A -85,B 0,C 180,E1 -11254.073,E2 -11254.073} C_VEL
LIN {X 0,Y 395.83,Z 396.742,A -85,B 0,C 180,E1 -11255.804,E2 -11255.804} C_VEL
LIN {X 0,Y 396.081,Z 391.682,A -85,B 0,C 180,E1 -11257.647,E2 -11257.647} C_VEL
LIN {X 0,Y 396.519,Z 385.18,A -85,B 0,C 180,E1 -11259.436,E2 -11259.436} C_VEL
LIN {X 0,Y 397.052,Z 378.1,A -85,B 0,C 180,E1 -11260.969,E2 -11260.969} C_VEL
LIN {X 0,Y 397.955,Z 369.275,A -85,B 0,C 180,E1 -11262.494,E2 -11262.494} C_VEL
LIN {X 0,Y 398.732,Z 359.176,A -85,B 0,C 180,E1 -11263.91,E2 -11263.91} C_VEL
LIN {X 0,Y 399.668,Z 348.001,A -85,B 0,C 180,E1 -11265.15,E2 -11265.15} C_VEL
LIN {X 0,Y 400.67,Z 336.426,A -85,B 0,C 180,E1 -11266.168,E2 -11266.168} C_VEL
LIN {X 0,Y 401.264,Z 327.8,A -85,B 0,C 180,E1 -11266.777,E2 -11266.777} C_VEL
LIN {X 0,Y 400.115,Z 316.192,A -85,B 0,C 180,E1 -11267.518,E2 -11267.518} C_VEL
LIN {X 0,Y 397.926,Z 303.624,A -85,B 0,C 180,E1 -11268.172,E2 -11268.172} C_VEL
LIN {X 0,Y 396.338,Z 296.044,A -85,B 0,C 180,E1 -11268.501,E2 -11268.501} C_VEL
LIN {X 0,Y 396.733,Z 288.339,A -85,B 0,C 180,E1 -11272.38,E2 -11272.38} C_VEL
LIN {X 0,Y 397.156,Z 280.924,A -85,B 0,C 180,E1 -11276.256,E2 -11276.256} C_VEL
LIN {X 0,Y 397.659,Z 274.086,A -85,B 0,C 180,E1 -11280.002,E2 -11280.002} C_VEL
LIN {X 0,Y 398.185,Z 268.504,A -85,B 0,C 180,E1 -11283.171,E2 -11283.171} C_VEL
LIN {X 0,Y 398.448,Z 266.48,A -85,B 0,C 180,E1 -11284.362,E2 -11284.362} C_VEL
LIN {X 0,Y 398.38,Z 262.509,A -85,B 0,C 180,E1 -11286.855,E2 -11286.855} C_VEL
LIN {X 0,Y 397.863,Z 258.65,A -85,B 0,C 180,E1 -11289.487,E2 -11289.487} C_VEL
LIN {X 0,Y 397.122,Z 254.02,A -85,B 0,C 180,E1 -11292.948,E2 -11292.948} C_VEL
LIN {X 0,Y 397.103,Z 254.022,A -85,B 0,C 180,E1 -11296.519,E2 -11296.519} C_VEL
LIN {X 0,Y 397.119,Z 254.023,A -85,B 0,C 180,E1 -11299.55,E2 -11299.55} C_VEL
LIN {X 0,Y 397.097,Z 254.024,A -85,B 0,C 180,E1 -11302.789,E2 -11302.789} C_VEL
LIN {X 0,Y 397.116,Z 254.02,A -85,B 0,C 180,E1 -11306.281,E2 -11306.281} C_VEL
LIN {X 0,Y 397.111,Z 254.021,A -85,B 0,C 180,E1 -11310.132,E2 -11310.132} C_VEL
LIN {X 0,Y 397.191,Z 254.01,A -85,B 0,C 180,E1 -11312.609,E2 -11312.609} C_VEL
LIN {X 0,Y 397.129,Z 254.019,A -85,B 0,C 180,E1 -11315.98,E2 -11315.98} C_VEL
LIN {X 0,Y 397.134,Z 254.018,A -85,B 0,C 180,E1 -11319.703,E2 -11319.703} C_VEL
LIN {X 0,Y 397.177,Z 254.012,A -85,B 0,C 180,E1 -11322.844,E2 -11322.844} C_VEL
LIN {X 0,Y 397.223,Z 254.007,A -85,B 0,C 180,E1 -11326.701,E2 -11326.701} C_VEL
LIN {X 0,Y 397.213,Z 254.008,A -85,B 0,C 180,E1 -11329.808,E2 -11329.808} C_VEL
LIN {X 0,Y 397.357,Z 253.991,A -85,B 0,C 180,E1 -11332.887,E2 -11332.887} C_VEL
LIN {X 0,Y 397.249,Z 254.002,A -85,B 0,C 180,E1 -11334.924,E2 -11334.924} C_VEL
LIN {X 0,Y 397.444,Z 253.979,A -85,B 0,C 180,E1 -11337.972,E2 -11337.972} C_VEL
LIN {X 0,Y 397.573,Z 253.963,A -85,B 0,C 180,E1 -11339.999,E2 -11339.999} C_VEL
LIN {X 0,Y 397.375,Z 253.991,A -85,B 0,C 180,E1 -11343.04,E2 -11343.04} C_VEL
LIN {X 0,Y 397.341,Z 253.991,A -85,B 0,C 180,E1 -11346.648,E2 -11346.648} C_VEL
LIN {X 0,Y 397.326,Z 253.996,A -85,B 0,C 180,E1 -11348.134,E2 -11348.134} C_VEL
LIN {X 0,Y 397.354,Z 257.26,A -85,B 0,C 180,E1 -11351.217,E2 -11351.217} C_VEL
LIN {X 0,Y 397.262,Z 259.638,A -85,B 0,C 180,E1 -11353.347,E2 -11353.347} C_VEL
LIN {X 0,Y 396.954,Z 263.98,A -85,B 0,C 180,E1 -11357.052,E2 -11357.052} C_VEL
LIN {X 0,Y 396.626,Z 268.504,A -85,B 0,C 180,E1 -11360.755,E2 -11360.755} C_VEL
LIN {X 0,Y 396.427,Z 272.668,A -85,B 0,C 180,E1 -11364.062,E2 -11364.062} C_VEL
LIN {X 0,Y 396.23,Z 277.215,A -85,B 0,C 180,E1 -11367.582,E2 -11367.582} C_VEL
LIN {X 0,Y 399.893,Z 291.581,A -85,B 0,C 180,E1 -11368.326,E2 -11368.326} C_VEL
LIN {X 0,Y 401.981,Z 303.076,A -85,B 0,C 180,E1 -11369.055,E2 -11369.055} C_VEL
LIN {X 0,Y 401.226,Z 315.06,A -85,B 0,C 180,E1 -11369.874,E2 -11369.874} C_VEL
LIN {X 0,Y 400.33,Z 326.67,A -85,B 0,C 180,E1 -11370.904,E2 -11370.904} C_VEL
LIN {X 0,Y 399.453,Z 337.306,A -85,B 0,C 180,E1 -11372.087,E2 -11372.087} C_VEL
LIN {X 0,Y 398.585,Z 346.345,A -85,B 0,C 180,E1 -11373.329,E2 -11373.329} C_VEL
LIN {X 0,Y 397.801,Z 354.451,A -85,B 0,C 180,E1 -11374.695,E2 -11374.695} C_VEL
LIN {X 0,Y 397.067,Z 362.425,A -85,B 0,C 180,E1 -11376.364,E2 -11376.364} C_VEL
LIN {X 0,Y 396.541,Z 368.662,A -85,B 0,C 180,E1 -11378.027,E2 -11378.027} C_VEL
LIN {X 0,Y 396.132,Z 373.452,A -85,B 0,C 180,E1 -11379.693,E2 -11379.693} C_VEL
LIN {X 0,Y 395.919,Z 376.453,A -85,B 0,C 180,E1 -11381.054,E2 -11381.054} C_VEL
LIN {X 0,Y 395.759,Z 378.659,A -85,B 0,C 180,E1 -11382.438,E2 -11382.438} C_VEL
LIN {X 0,Y 395.665,Z 380.124,A -85,B 0,C 180,E1 -11383.845,E2 -11383.845} C_VEL
LIN {X 0,Y 395.59,Z 380.843,A -85,B 0,C 180,E1 -11385.284,E2 -11385.284} C_VEL
LIN {X 0,Y 395.545,Z 380.761,A -85,B 0,C 180,E1 -11386.757,E2 -11386.757} C_VEL
LIN {X 0,Y 395.614,Z 379.798,A -85,B 0,C 180,E1 -11388.253,E2 -11388.253} C_VEL
LIN {X 0,Y 395.751,Z 377.11,A -85,B 0,C 180,E1 -11390.261,E2 -11390.261} C_VEL
LIN {X 0,Y 395.975,Z 374.423,A -85,B 0,C 180,E1 -11391.597,E2 -11391.597} C_VEL
LIN {X 0,Y 396.221,Z 370.85,A -85,B 0,C 180,E1 -11392.955,E2 -11392.955} C_VEL
LIN {X 0,Y 396.6,Z 365.311,A -85,B 0,C 180,E1 -11394.599,E2 -11394.599} C_VEL
LIN {X 0,Y 397.133,Z 358.048,A -85,B 0,C 180,E1 -11396.276,E2 -11396.276} C_VEL
LIN {X 0,Y 397.782,Z 350.397,A -85,B 0,C 180,E1 -11397.694,E2 -11397.694} C_VEL
LIN {X 0,Y 398.519,Z 341.105,A -85,B 0,C 180,E1 -11399.095,E2 -11399.095} C_VEL
LIN {X 0,Y 399.272,Z 330.786,A -85,B 0,C 180,E1 -11400.343,E2 -11400.343} C_VEL
LIN {X 0,Y 400.102,Z 319.572,A -85,B 0,C 180,E1 -11401.432,E2 -11401.432} C_VEL
LIN {X 0,Y 400.77,Z 308.091,A -85,B 0,C 180,E1 -11402.309,E2 -11402.309} C_VEL
LIN {X 0,Y 401.019,Z 300.974,A -85,B 0,C 180,E1 -11402.752,E2 -11402.752} C_VEL
LIN {X 0,Y 398.648,Z 288.105,A -85,B 0,C 180,E1 -11403.497,E2 -11403.497} C_VEL
LIN {X 0,Y 396.075,Z 276.398,A -85,B 0,C 180,E1 -11404.021,E2 -11404.021} C_VEL
LIN {X 0,Y 396.246,Z 271.98,A -85,B 0,C 180,E1 -11407.26,E2 -11407.26} C_VEL
LIN {X 0,Y 396.431,Z 267.881,A -85,B 0,C 180,E1 -11410.316,E2 -11410.316} C_VEL
LIN {X 0,Y 396.612,Z 263.66,A -85,B 0,C 180,E1 -11413.53,E2 -11413.53} C_VEL
LIN {X 0,Y 396.897,Z 258.263,A -85,B 0,C 180,E1 -11417.732,E2 -11417.732} C_VEL
LIN {X 0,Y 397.019,Z 254.411,A -85,B 0,C 180,E1 -11420.833,E2 -11420.833} C_VEL
LIN {X 0,Y 397.214,Z 254.005,A -85,B 0,C 180,E1 -11422.218,E2 -11422.218} C_VEL
LIN {X 0,Y 397.346,Z 253.989,A -85,B 0,C 180,E1 -11423.908,E2 -11423.908} C_VEL
LIN {X 0,Y 397.441,Z 253.977,A -85,B 0,C 180,E1 -11427.973,E2 -11427.973} C_VEL
LIN {X 0,Y 397.572,Z 253.962,A -85,B 0,C 180,E1 -11430,E2 -11430} C_VEL
LIN {X 0,Y 397.372,Z 253.987,A -85,B 0,C 180,E1 -11433.042,E2 -11433.042} C_VEL
LIN {X 0,Y 397.353,Z 253.988,A -85,B 0,C 180,E1 -11437.112,E2 -11437.112} C_VEL
LIN {X 0,Y 397.219,Z 254.008,A -85,B 0,C 180,E1 -11440.191,E2 -11440.191} C_VEL
LIN {X 0,Y 397.197,Z 254.007,A -85,B 0,C 180,E1 -11441.287,E2 -11441.287} C_VEL
LIN {X 0,Y 396.521,Z 254.095,A -85,B 0,C 180,E1 -11442.133,E2 -11442.133} C_VEL
LIN {X 0,Y 393.682,Z 254.449,A -85,B 0,C 180,E1 -11443.508,E2 -11443.508} C_VEL
LIN {X 0,Y 391.274,Z 254.751,A -85,B 0,C 180,E1 -11444.619,E2 -11444.619} C_VEL
LIN {X 0,Y 390.223,Z 254.879,A -85,B 0,C 180,E1 -11445.477,E2 -11445.477} C_VEL
LIN {X 0,Y 390.128,Z 254.889,A -85,B 0,C 180,E1 -11445.768,E2 -11445.768} C_VEL
LIN {X 0,Y 390.106,Z 254.89,A -85,B 0,C 180,E1 -11448.922,E2 -11448.922} C_VEL
LIN {X 0,Y 390.052,Z 254.9,A -85,B 0,C 180,E1 -11452.233,E2 -11452.233} C_VEL
LIN {X 0,Y 390.108,Z 254.893,A -85,B 0,C 180,E1 -11455.744,E2 -11455.744} C_VEL
LIN {X 0,Y 390.054,Z 254.897,A -85,B 0,C 180,E1 -11459.109,E2 -11459.109} C_VEL
LIN {X 0,Y 390.044,Z 254.897,A -85,B 0,C 180,E1 -11462.721,E2 -11462.721} C_VEL
LIN {X 0,Y 390.047,Z 254.901,A -85,B 0,C 180,E1 -11465.826,E2 -11465.826} C_VEL
LIN {X 0,Y 390.064,Z 254.898,A -85,B 0,C 180,E1 -11469.22,E2 -11469.22} C_VEL
LIN {X 0,Y 390.112,Z 254.889,A -85,B 0,C 180,E1 -11472.388,E2 -11472.388} C_VEL
LIN {X 0,Y 390.107,Z 254.895,A -85,B 0,C 180,E1 -11475.366,E2 -11475.366} C_VEL
LIN {X 0,Y 390.094,Z 254.891,A -85,B 0,C 180,E1 -11478.197,E2 -11478.197} C_VEL
LIN {X 0,Y 390.085,Z 254.895,A -85,B 0,C 180,E1 -11480.909,E2 -11480.909} C_VEL
LIN {X 0,Y 390.076,Z 254.896,A -85,B 0,C 180,E1 -11484.794,E2 -11484.794} C_VEL
LIN {X 0,Y 390.018,Z 254.902,A -85,B 0,C 180,E1 -11488.497,E2 -11488.497} C_VEL
LIN {X 0,Y 390.108,Z 254.89,A -85,B 0,C 180,E1 -11492.071,E2 -11492.071} C_VEL
LIN {X 0,Y 390.071,Z 254.896,A -85,B 0,C 180,E1 -11495.52,E2 -11495.52} C_VEL
LIN {X 0,Y 390.047,Z 254.902,A -85,B 0,C 180,E1 -11498.879,E2 -11498.879} C_VEL
LIN {X 0,Y 390.12,Z 254.89,A -85,B 0,C 180,E1 -11502.168,E2 -11502.168} C_VEL
LIN {X 0,Y 390.136,Z 254.887,A -85,B 0,C 180,E1 -11505.394,E2 -11505.394} C_VEL
LIN {X 0,Y 390.142,Z 254.89,A -85,B 0,C 180,E1 -11508.572,E2 -11508.572} C_VEL
LIN {X 0,Y 390.301,Z 254.868,A -85,B 0,C 180,E1 -11512.033,E2 -11512.033} C_VEL
LIN {X 0,Y 390.22,Z 254.878,A -85,B 0,C 180,E1 -11514.835,E2 -11514.835} C_VEL
LIN {X 0,Y 390.414,Z 254.855,A -85,B 0,C 180,E1 -11517.938,E2 -11517.938} C_VEL
LIN {X 0,Y 390.544,Z 254.84,A -85,B 0,C 180,E1 -11520.001,E2 -11520.001} C_VEL
LIN {X 0,Y 390.31,Z 254.865,A -85,B 0,C 180,E1 -11523.098,E2 -11523.098} C_VEL
LIN {X 0,Y 390.325,Z 254.867,A -85,B 0,C 180,E1 -11526.203,E2 -11526.203} C_VEL
LIN {X 0,Y 390.311,Z 254.868,A -85,B 0,C 180,E1 -11528.283,E2 -11528.283} C_VEL
LIN {X 0,Y 390.174,Z 254.883,A -85,B 0,C 180,E1 -11532.484,E2 -11532.484} C_VEL
LIN {X 0,Y 390.136,Z 254.89,A -85,B 0,C 180,E1 -11535.678,E2 -11535.678} C_VEL
LIN {X 0,Y 390.102,Z 254.891,A -85,B 0,C 180,E1 -11538.923,E2 -11538.923} C_VEL
LIN {X 0,Y 390.037,Z 254.9,A -85,B 0,C 180,E1 -11542.235,E2 -11542.235} C_VEL
LIN {X 0,Y 390.117,Z 254.893,A -85,B 0,C 180,E1 -11545.745,E2 -11545.745} C_VEL
LIN {X 0,Y 390.057,Z 254.899,A -85,B 0,C 180,E1 -11549.111,E2 -11549.111} C_VEL
LIN {X 0,Y 390.042,Z 254.899,A -85,B 0,C 180,E1 -11552.723,E2 -11552.723} C_VEL
LIN {X 0,Y 390.056,Z 254.898,A -85,B 0,C 180,E1 -11555.826,E2 -11555.826} C_VEL
LIN {X 0,Y 390.071,Z 254.899,A -85,B 0,C 180,E1 -11559.22,E2 -11559.22} C_VEL
LIN {X 0,Y 390.042,Z 254.898,A -85,B 0,C 180,E1 -11562.375,E2 -11562.375} C_VEL
LIN {X 0,Y 390.045,Z 254.901,A -85,B 0,C 180,E1 -11565.355,E2 -11565.355} C_VEL
LIN {X 0,Y 390.108,Z 255.072,A -85,B 0,C 180,E1 -11568.852,E2 -11568.852} C_VEL
LIN {X 0,Y 390.876,Z 259.529,A -85,B 0,C 180,E1 -11571.662,E2 -11571.662} C_VEL
LIN {X 0,Y 391.282,Z 263.292,A -85,B 0,C 180,E1 -11573.928,E2 -11573.928} C_VEL
LIN {X 0,Y 391.141,Z 268.245,A -85,B 0,C 180,E1 -11576.769,E2 -11576.769} C_VEL
LIN {X 0,Y 390.502,Z 274.766,A -85,B 0,C 180,E1 -11580.336,E2 -11580.336} C_VEL
LIN {X 0,Y 389.957,Z 282.356,A -85,B 0,C 180,E1 -11584.371,E2 -11584.371} C_VEL
LIN {X 0,Y 389.618,Z 288.856,A -85,B 0,C 180,E1 -11587.741,E2 -11587.741} C_VEL
LIN {X 0,Y 389.279,Z 295.35,A -85,B 0,C 180,E1 -11591.036,E2 -11591.036} C_VEL
LIN {X 0,Y 389.239,Z 296.633,A -85,B 0,C 180,E1 -11591.683,E2 -11591.683} C_VEL
LIN {X 0,Y 391.975,Z 312.538,A -85,B 0,C 180,E1 -11592.385,E2 -11592.385} C_VEL
LIN {X 0,Y 393.585,Z 325.354,A -85,B 0,C 180,E1 -11593.139,E2 -11593.139} C_VEL
LIN {X 0,Y 393.603,Z 331.172,A -85,B 0,C 180,E1 -11593.534,E2 -11593.534} C_VEL
LIN {X 0,Y 392.731,Z 342.484,A -85,B 0,C 180,E1 -11594.429,E2 -11594.429} C_VEL
LIN {X 0,Y 391.871,Z 352.854,A -85,B 0,C 180,E1 -11595.459,E2 -11595.459} C_VEL
LIN {X 0,Y 391.088,Z 363.37,A -85,B 0,C 180,E1 -11596.755,E2 -11596.755} C_VEL
LIN {X 0,Y 390.409,Z 371.892,A -85,B 0,C 180,E1 -11598.052,E2 -11598.052} C_VEL
LIN {X 0,Y 389.712,Z 380.198,A -85,B 0,C 180,E1 -11599.611,E2 -11599.611} C_VEL
LIN {X 0,Y 389.259,Z 386.894,A -85,B 0,C 180,E1 -11601.172,E2 -11601.172} C_VEL
LIN {X 0,Y 388.939,Z 392.23,A -85,B 0,C 180,E1 -11602.733,E2 -11602.733} C_VEL
LIN {X 0,Y 388.729,Z 396.264,A -85,B 0,C 180,E1 -11604.248,E2 -11604.248} C_VEL
LIN {X 0,Y 388.701,Z 399.447,A -85,B 0,C 180,E1 -11605.853,E2 -11605.853} C_VEL
LIN {X 0,Y 388.638,Z 400.963,A -85,B 0,C 180,E1 -11606.89,E2 -11606.89} C_VEL
LIN {X 0,Y 388.664,Z 402.022,A -85,B 0,C 180,E1 -11607.927,E2 -11607.927} C_VEL
LIN {X 0,Y 388.704,Z 402.682,A -85,B 0,C 180,E1 -11608.964,E2 -11608.964} C_VEL
LIN {X 0,Y 388.709,Z 402.949,A -85,B 0,C 180,E1 -11610,E2 -11610} C_VEL
LIN {X 0,Y 388.704,Z 402.816,A -85,B 0,C 180,E1 -11611.036,E2 -11611.036} C_VEL
LIN {X 0,Y 388.662,Z 402.242,A -85,B 0,C 180,E1 -11612.072,E2 -11612.072} C_VEL
LIN {X 0,Y 388.701,Z 399.906,A -85,B 0,C 180,E1 -11614.147,E2 -11614.147} C_VEL
LIN {X 0,Y 388.73,Z 396.928,A -85,B 0,C 180,E1 -11615.753,E2 -11615.753} C_VEL
LIN {X 0,Y 388.94,Z 393.117,A -85,B 0,C 180,E1 -11617.266,E2 -11617.266} C_VEL
LIN {X 0,Y 389.269,Z 388.079,A -85,B 0,C 180,E1 -11618.827,E2 -11618.827} C_VEL
LIN {X 0,Y 389.813,Z 381.766,A -85,B 0,C 180,E1 -11620.386,E2 -11620.386} C_VEL
LIN {X 0,Y 390.502,Z 373.89,A -85,B 0,C 180,E1 -11621.944,E2 -11621.944} C_VEL
LIN {X 0,Y 391.491,Z 364.096,A -85,B 0,C 180,E1 -11623.495,E2 -11623.495} C_VEL
LIN {X 0,Y 392.281,Z 354.212,A -85,B 0,C 180,E1 -11624.764,E2 -11624.764} C_VEL
LIN {X 0,Y 393.337,Z 342.596,A -85,B 0,C 180,E1 -11625.945,E2 -11625.945} C_VEL
LIN {X 0,Y 394.401,Z 329.998,A -85,B 0,C 180,E1 -11626.945,E2 -11626.945} C_VEL
LIN {X 0,Y 393.909,Z 321.904,A -85,B 0,C 180,E1 -11627.502,E2 -11627.502} C_VEL
LIN {X 0,Y 391.989,Z 308.626,A -85,B 0,C 180,E1 -11628.291,E2 -11628.291} C_VEL
LIN {X 0,Y 389.29,Z 295.842,A -85,B 0,C 180,E1 -11628.896,E2 -11628.896} C_VEL
LIN {X 0,Y 389.653,Z 289.298,A -85,B 0,C 180,E1 -11632.257,E2 -11632.257} C_VEL
LIN {X 0,Y 390.01,Z 282.804,A -85,B 0,C 180,E1 -11635.708,E2 -11635.708} C_VEL
LIN {X 0,Y 390.459,Z 276.719,A -85,B 0,C 180,E1 -11639.076,E2 -11639.076} C_VEL
LIN {X 0,Y 391.069,Z 270.541,A -85,B 0,C 180,E1 -11642.624,E2 -11642.624} C_VEL
LIN {X 0,Y 391.452,Z 266.534,A -85,B 0,C 180,E1 -11645.065,E2 -11645.065} C_VEL
LIN {X 0,Y 391.232,Z 262.406,A -85,B 0,C 180,E1 -11647.775,E2 -11647.775} C_VEL
LIN {X 0,Y 390.572,Z 258.043,A -85,B 0,C 180,E1 -11650.908,E2 -11650.908} C_VEL
LIN {X 0,Y 390.059,Z 254.9,A -85,B 0,C 180,E1 -11653.5,E2 -11653.5} C_VEL
LIN {X 0,Y 390.066,Z 254.9,A -85,B 0,C 180,E1 -11656.79,E2 -11656.79} C_VEL
LIN {X 0,Y 390.074,Z 254.901,A -85,B 0,C 180,E1 -11659.562,E2 -11659.562} C_VEL
LIN {X 0,Y 390.045,Z 254.903,A -85,B 0,C 180,E1 -11662.447,E2 -11662.447} C_VEL
LIN {X 0,Y 390.066,Z 254.899,A -85,B 0,C 180,E1 -11666.044,E2 -11666.044} C_VEL
LIN {X 0,Y 390.049,Z 254.9,A -85,B 0,C 180,E1 -11669.866,E2 -11669.866} C_VEL
LIN {X 0,Y 390.11,Z 254.892,A -85,B 0,C 180,E1 -11673.23,E2 -11673.23} C_VEL
LIN {X 0,Y 390.102,Z 254.894,A -85,B 0,C 180,E1 -11676.749,E2 -11676.749} C_VEL
LIN {X 0,Y 390.099,Z 254.895,A -85,B 0,C 180,E1 -11679.982,E2 -11679.982} C_VEL
LIN {X 0,Y 390.133,Z 254.891,A -85,B 0,C 180,E1 -11683.247,E2 -11683.247} C_VEL
LIN {X 0,Y 390.189,Z 254.883,A -85,B 0,C 180,E1 -11686.56,E2 -11686.56} C_VEL
LIN {X 0,Y 390.163,Z 254.887,A -85,B 0,C 180,E1 -11689.622,E2 -11689.622} C_VEL
LIN {X 0,Y 390.312,Z 254.868,A -85,B 0,C 180,E1 -11692.758,E2 -11692.758} C_VEL
LIN {X 0,Y 390.221,Z 254.877,A -85,B 0,C 180,E1 -11694.832,E2 -11694.832} C_VEL
LIN {X 0,Y 390.413,Z 254.855,A -85,B 0,C 180,E1 -11697.936,E2 -11697.936} C_VEL
LIN {X 0,Y 390.542,Z 254.839,A -85,B 0,C 180,E1 -11699.999,E2 -11699.999} C_VEL
LIN {X 0,Y 390.309,Z 254.871,A -85,B 0,C 180,E1 -11703.095,E2 -11703.095} C_VEL
LIN {X 0,Y 390.295,Z 254.869,A -85,B 0,C 180,E1 -11706.644,E2 -11706.644} C_VEL
LIN {X 0,Y 390.327,Z 254.999,A -85,B 0,C 180,E1 -11707.997,E2 -11707.997} C_VEL
LIN {X 0,Y 390.32,Z 258.576,A -85,B 0,C 180,E1 -11711.422,E2 -11711.422} C_VEL
LIN {X 0,Y 390.082,Z 262.112,A -85,B 0,C 180,E1 -11714.608,E2 -11714.608} C_VEL
LIN {X 0,Y 389.834,Z 265.893,A -85,B 0,C 180,E1 -11717.846,E2 -11717.846} C_VEL
LIN {X 0,Y 389.536,Z 269.869,A -85,B 0,C 180,E1 -11721.15,E2 -11721.15} C_VEL
LIN {X 0,Y 389.32,Z 274.069,A -85,B 0,C 180,E1 -11724.53,E2 -11724.53} C_VEL
LIN {X 0,Y 389.161,Z 277.429,A -85,B 0,C 180,E1 -11727.182,E2 -11727.182} C_VEL
LIN {X 0,Y 392.774,Z 291.229,A -85,B 0,C 180,E1 -11727.923,E2 -11727.923} C_VEL
LIN {X 0,Y 395.107,Z 303.06,A -85,B 0,C 180,E1 -11728.701,E2 -11728.701} C_VEL
LIN {X 0,Y 394.608,Z 313.4,A -85,B 0,C 180,E1 -11729.415,E2 -11729.415} C_VEL
LIN {X 0,Y 393.676,Z 325.187,A -85,B 0,C 180,E1 -11730.433,E2 -11730.433} C_VEL
LIN {X 0,Y 392.773,Z 335.474,A -85,B 0,C 180,E1 -11731.557,E2 -11731.557} C_VEL
LIN {X 0,Y 391.838,Z 345.127,A -85,B 0,C 180,E1 -11732.856,E2 -11732.856} C_VEL
LIN {X 0,Y 390.9,Z 354.324,A -85,B 0,C 180,E1 -11734.394,E2 -11734.394} C_VEL
LIN {X 0,Y 390.085,Z 362.535,A -85,B 0,C 180,E1 -11736.134,E2 -11736.134} C_VEL
LIN {X 0,Y 389.529,Z 368.83,A -85,B 0,C 180,E1 -11737.837,E2 -11737.837} C_VEL
LIN {X 0,Y 389.188,Z 372.788,A -85,B 0,C 180,E1 -11739.198,E2 -11739.198} C_VEL
LIN {X 0,Y 388.793,Z 377.256,A -85,B 0,C 180,E1 -11741.281,E2 -11741.281} C_VEL
LIN {X 0,Y 388.707,Z 378.61,A -85,B 0,C 180,E1 -11742.159,E2 -11742.159} C_VEL
LIN {X 0,Y 388.587,Z 380.241,A -85,B 0,C 180,E1 -11743.662,E2 -11743.662} C_VEL
LIN {X 0,Y 388.51,Z 381.029,A -85,B 0,C 180,E1 -11745.132,E2 -11745.132} C_VEL
LIN {X 0,Y 388.456,Z 381.007,A -85,B 0,C 180,E1 -11746.569,E2 -11746.569} C_VEL
LIN {X 0,Y 388.515,Z 380.219,A -85,B 0,C 180,E1 -11747.988,E2 -11747.988} C_VEL
LIN {X 0,Y 388.666,Z 377.693,A -85,B 0,C 180,E1 -11750.089,E2 -11750.089} C_VEL
LIN {X 0,Y 388.874,Z 374.881,A -85,B 0,C 180,E1 -11751.556,E2 -11751.556} C_VEL
LIN {X 0,Y 389.247,Z 369.902,A -85,B 0,C 180,E1 -11753.429,E2 -11753.429} C_VEL
LIN {X 0,Y 389.674,Z 364.169,A -85,B 0,C 180,E1 -11755.067,E2 -11755.067} C_VEL
LIN {X 0,Y 390.253,Z 357.036,A -85,B 0,C 180,E1 -11756.684,E2 -11756.684} C_VEL
LIN {X 0,Y 391.007,Z 348.063,A -85,B 0,C 180,E1 -11758.292,E2 -11758.292} C_VEL
LIN {X 0,Y 391.775,Z 338.583,A -85,B 0,C 180,E1 -11759.66,E2 -11759.66} C_VEL
LIN {X 0,Y 392.511,Z 328.913,A -85,B 0,C 180,E1 -11760.797,E2 -11760.797} C_VEL
LIN {X 0,Y 393.347,Z 317.297,A -85,B 0,C 180,E1 -11761.885,E2 -11761.885} C_VEL
LIN {X 0,Y 394.149,Z 305.079,A -85,B 0,C 180,E1 -11762.777,E2 -11762.777} C_VEL
LIN {X 0,Y 394.049,Z 301.473,A -85,B 0,C 180,E1 -11763.006,E2 -11763.006} C_VEL
LIN {X 0,Y 391.699,Z 288.644,A -85,B 0,C 180,E1 -11763.765,E2 -11763.765} C_VEL
LIN {X 0,Y 389.007,Z 276.573,A -85,B 0,C 180,E1 -11764.331,E2 -11764.331} C_VEL
LIN {X 0,Y 389.18,Z 272.027,A -85,B 0,C 180,E1 -11767.715,E2 -11767.715} C_VEL
LIN {X 0,Y 389.363,Z 269.081,A -85,B 0,C 180,E1 -11769.944,E2 -11769.944} C_VEL
LIN {X 0,Y 389.525,Z 264.823,A -85,B 0,C 180,E1 -11773.222,E2 -11773.222} C_VEL
LIN {X 0,Y 389.828,Z 259.388,A -85,B 0,C 180,E1 -11777.506,E2 -11777.506} C_VEL
LIN {X 0,Y 389.983,Z 255.501,A -85,B 0,C 180,E1 -11780.666,E2 -11780.666} C_VEL
LIN {X 0,Y 390.164,Z 254.883,A -85,B 0,C 180,E1 -11782.171,E2 -11782.171} C_VEL
LIN {X 0,Y 390.295,Z 254.867,A -85,B 0,C 180,E1 -11783.798,E2 -11783.798} C_VEL
LIN {X 0,Y 390.41,Z 254.853,A -85,B 0,C 180,E1 -11787.937,E2 -11787.937} C_VEL
LIN {X 0,Y 390.541,Z 254.838,A -85,B 0,C 180,E1 -11790,E2 -11790} C_VEL
LIN {X 0,Y 390.306,Z 254.866,A -85,B 0,C 180,E1 -11793.097,E2 -11793.097} C_VEL
LIN {X 0,Y 390.32,Z 254.867,A -85,B 0,C 180,E1 -11796.202,E2 -11796.202} C_VEL
LIN {X 0,Y 390.304,Z 254.87,A -85,B 0,C 180,E1 -11798.282,E2 -11798.282} C_VEL
LIN {X 0,Y 390.167,Z 254.886,A -85,B 0,C 180,E1 -11802.483,E2 -11802.483} C_VEL
LIN {X 0,Y 390.128,Z 254.889,A -85,B 0,C 180,E1 -11805.768,E2 -11805.768} C_VEL
LIN {X 0,Y 389.425,Z 254.977,A -85,B 0,C 180,E1 -11806.63,E2 -11806.63} C_VEL
LIN {X 0,Y 386.535,Z 255.339,A -85,B 0,C 180,E1 -11808.029,E2 -11808.029} C_VEL
LIN {X 0,Y 384.126,Z 255.635,A -85,B 0,C 180,E1 -11809.16,E2 -11809.16} C_VEL
LIN {X 0,Y 383.123,Z 255.765,A -85,B 0,C 180,E1 -11810.035,E2 -11810.035} C_VEL
LIN {X 0,Y 383.057,Z 255.77,A -85,B 0,C 180,E1 -11810.332,E2 -11810.332} C_VEL
LIN {X 0,Y 383.032,Z 255.776,A -85,B 0,C 180,E1 -11813.807,E2 -11813.807} C_VEL
LIN {X 0,Y 383.046,Z 255.771,A -85,B 0,C 180,E1 -11817.302,E2 -11817.302} C_VEL
LIN {X 0,Y 382.985,Z 255.777,A -85,B 0,C 180,E1 -11820.918,E2 -11820.918} C_VEL
LIN {X 0,Y 383.007,Z 255.775,A -85,B 0,C 180,E1 -11824.341,E2 -11824.341} C_VEL
LIN {X 0,Y 382.988,Z 255.78,A -85,B 0,C 180,E1 -11827.269,E2 -11827.269} C_VEL
LIN {X 0,Y 383.01,Z 255.776,A -85,B 0,C 180,E1 -11829.957,E2 -11829.957} C_VEL
LIN {X 0,Y 383.055,Z 255.769,A -85,B 0,C 180,E1 -11832.789,E2 -11832.789} C_VEL
LIN {X 0,Y 383.059,Z 255.77,A -85,B 0,C 180,E1 -11835.801,E2 -11835.801} C_VEL
LIN {X 0,Y 383.034,Z 255.772,A -85,B 0,C 180,E1 -11838.787,E2 -11838.787} C_VEL
LIN {X 0,Y 382.993,Z 255.776,A -85,B 0,C 180,E1 -11842.096,E2 -11842.096} C_VEL
LIN {X 0,Y 383.008,Z 255.778,A -85,B 0,C 180,E1 -11845.333,E2 -11845.333} C_VEL
LIN {X 0,Y 382.977,Z 255.782,A -85,B 0,C 180,E1 -11849.083,E2 -11849.083} C_VEL
LIN {X 0,Y 383.048,Z 255.773,A -85,B 0,C 180,E1 -11852.699,E2 -11852.699} C_VEL
LIN {X 0,Y 383.043,Z 255.774,A -85,B 0,C 180,E1 -11855.041,E2 -11855.041} C_VEL
LIN {X 0,Y 382.984,Z 255.78,A -85,B 0,C 180,E1 -11858.47,E2 -11858.47} C_VEL
LIN {X 0,Y 383.055,Z 255.769,A -85,B 0,C 180,E1 -11861.828,E2 -11861.828} C_VEL
LIN {X 0,Y 383.102,Z 255.764,A -85,B 0,C 180,E1 -11865.119,E2 -11865.119} C_VEL
LIN {X 0,Y 383.091,Z 255.768,A -85,B 0,C 180,E1 -11868.359,E2 -11868.359} C_VEL
LIN {X 0,Y 383.257,Z 255.745,A -85,B 0,C 180,E1 -11871.977,E2 -11871.977} C_VEL
LIN {X 0,Y 383.192,Z 255.754,A -85,B 0,C 180,E1 -11874.74,E2 -11874.74} C_VEL
LIN {X 0,Y 383.381,Z 255.73,A -85,B 0,C 180,E1 -11877.9,E2 -11877.9} C_VEL
LIN {X 0,Y 383.513,Z 255.715,A -85,B 0,C 180,E1 -11880.001,E2 -11880.001} C_VEL
LIN {X 0,Y 383.247,Z 255.745,A -85,B 0,C 180,E1 -11883.155,E2 -11883.155} C_VEL
LIN {X 0,Y 383.282,Z 255.744,A -85,B 0,C 180,E1 -11886.318,E2 -11886.318} C_VEL
LIN {X 0,Y 383.257,Z 255.746,A -85,B 0,C 180,E1 -11888.437,E2 -11888.437} C_VEL
LIN {X 0,Y 383.103,Z 255.765,A -85,B 0,C 180,E1 -11891.643,E2 -11891.643} C_VEL
LIN {X 0,Y 383.108,Z 255.762,A -85,B 0,C 180,E1 -11894.883,E2 -11894.883} C_VEL
LIN {X 0,Y 383.06,Z 255.77,A -85,B 0,C 180,E1 -11898.175,E2 -11898.175} C_VEL
LIN {X 0,Y 382.99,Z 255.781,A -85,B 0,C 180,E1 -11901.532,E2 -11901.532} C_VEL
LIN {X 0,Y 383.05,Z 255.77,A -85,B 0,C 180,E1 -11904.962,E2 -11904.962} C_VEL
LIN {X 0,Y 383.028,Z 255.772,A -85,B 0,C 180,E1 -11908.271,E2 -11908.271} C_VEL
LIN {X 0,Y 383.008,Z 255.775,A -85,B 0,C 180,E1 -11912.151,E2 -11912.151} C_VEL
LIN {X 0,Y 383.017,Z 255.774,A -85,B 0,C 180,E1 -11914.669,E2 -11914.669} C_VEL
LIN {X 0,Y 383.001,Z 255.776,A -85,B 0,C 180,E1 -11917.905,E2 -11917.905} C_VEL
LIN {X 0,Y 382.984,Z 255.781,A -85,B 0,C 180,E1 -11921.349,E2 -11921.349} C_VEL
LIN {X 0,Y 382.996,Z 255.776,A -85,B 0,C 180,E1 -11924.304,E2 -11924.304} C_VEL
LIN {X 0,Y 382.996,Z 255.779,A -85,B 0,C 180,E1 -11927.951,E2 -11927.951} C_VEL
LIN {X 0,Y 383.05,Z 255.989,A -85,B 0,C 180,E1 -11928.662,E2 -11928.662} C_VEL
LIN {X 0,Y 383.93,Z 261.066,A -85,B 0,C 180,E1 -11931.92,E2 -11931.92} C_VEL
LIN {X 0,Y 384.258,Z 264.779,A -85,B 0,C 180,E1 -11934.178,E2 -11934.178} C_VEL
LIN {X 0,Y 384.113,Z 269.126,A -85,B 0,C 180,E1 -11936.709,E2 -11936.709} C_VEL
LIN {X 0,Y 383.437,Z 275.61,A -85,B 0,C 180,E1 -11940.339,E2 -11940.339} C_VEL
LIN {X 0,Y 382.92,Z 282.508,A -85,B 0,C 180,E1 -11944.072,E2 -11944.072} C_VEL
LIN {X 0,Y 382.525,Z 289.695,A -85,B 0,C 180,E1 -11947.875,E2 -11947.875} C_VEL
LIN {X 0,Y 382.185,Z 296.493,A -85,B 0,C 180,E1 -11951.393,E2 -11951.393} C_VEL
LIN {X 0,Y 384.599,Z 310.151,A -85,B 0,C 180,E1 -11951.979,E2 -11951.979} C_VEL
LIN {X 0,Y 386.375,Z 323.616,A -85,B 0,C 180,E1 -11952.763,E2 -11952.763} C_VEL
LIN {X 0,Y 386.849,Z 328.488,A -85,B 0,C 180,E1 -11953.102,E2 -11953.102} C_VEL
LIN {X 0,Y 385.98,Z 340.43,A -85,B 0,C 180,E1 -11954.014,E2 -11954.014} C_VEL
LIN {X 0,Y 385.077,Z 351.153,A -85,B 0,C 180,E1 -11955.061,E2 -11955.061} C_VEL
LIN {X 0,Y 384.287,Z 360.945,A -85,B 0,C 180,E1 -11956.246,E2 -11956.246} C_VEL
LIN {X 0,Y 383.579,Z 369.876,A -85,B 0,C 180,E1 -11957.568,E2 -11957.568} C_VEL
LIN {X 0,Y 382.753,Z 378.591,A -85,B 0,C 180,E1 -11959.152,E2 -11959.152} C_VEL
LIN {X 0,Y 382.254,Z 385.547,A -85,B 0,C 180,E1 -11960.742,E2 -11960.742} C_VEL
LIN {X 0,Y 381.867,Z 391.929,A -85,B 0,C 180,E1 -11962.598,E2 -11962.598} C_VEL
LIN {X 0,Y 381.69,Z 395.378,A -85,B 0,C 180,E1 -11963.882,E2 -11963.882} C_VEL
LIN {X 0,Y 381.626,Z 399.194,A -85,B 0,C 180,E1 -11965.775,E2 -11965.775} C_VEL
LIN {X 0,Y 381.549,Z 400.724,A -85,B 0,C 180,E1 -11966.832,E2 -11966.832} C_VEL
LIN {X 0,Y 381.563,Z 401.797,A -85,B 0,C 180,E1 -11967.889,E2 -11967.889} C_VEL
LIN {X 0,Y 381.619,Z 402.467,A -85,B 0,C 180,E1 -11968.945,E2 -11968.945} C_VEL
LIN {X 0,Y 381.64,Z 402.743,A -85,B 0,C 180,E1 -11970,E2 -11970} C_VEL
LIN {X 0,Y 381.604,Z 402.623,A -85,B 0,C 180,E1 -11971.055,E2 -11971.055} C_VEL
LIN {X 0,Y 381.56,Z 402.064,A -85,B 0,C 180,E1 -11972.111,E2 -11972.111} C_VEL
LIN {X 0,Y 381.626,Z 399.749,A -85,B 0,C 180,E1 -11974.224,E2 -11974.224} C_VEL
LIN {X 0,Y 381.673,Z 396.301,A -85,B 0,C 180,E1 -11976.093,E2 -11976.093} C_VEL
LIN {X 0,Y 381.98,Z 391.459,A -85,B 0,C 180,E1 -11977.931,E2 -11977.931} C_VEL
LIN {X 0,Y 382.482,Z 385.008,A -85,B 0,C 180,E1 -11979.786,E2 -11979.786} C_VEL
LIN {X 0,Y 383.076,Z 377.997,A -85,B 0,C 180,E1 -11981.374,E2 -11981.374} C_VEL
LIN {X 0,Y 384.048,Z 369.239,A -85,B 0,C 180,E1 -11982.954,E2 -11982.954} C_VEL
LIN {X 0,Y 384.913,Z 359.164,A -85,B 0,C 180,E1 -11984.428,E2 -11984.428} C_VEL
LIN {X 0,Y 385.877,Z 349.37,A -85,B 0,C 180,E1 -11985.583,E2 -11985.583} C_VEL
LIN {X 0,Y 386.926,Z 338.381,A -85,B 0,C 180,E1 -11986.623,E2 -11986.623} C_VEL
LIN {X 0,Y 387.607,Z 328.587,A -85,B 0,C 180,E1 -11987.377,E2 -11987.377} C_VEL
LIN {X 0,Y 386.305,Z 316.156,A -85,B 0,C 180,E1 -11988.228,E2 -11988.228} C_VEL
LIN {X 0,Y 383.978,Z 303.413,A -85,B 0,C 180,E1 -11988.943,E2 -11988.943} C_VEL
LIN {X 0,Y 382.256,Z 295.585,A -85,B 0,C 180,E1 -11989.325,E2 -11989.325} C_VEL
LIN {X 0,Y 382.615,Z 289.21,A -85,B 0,C 180,E1 -11992.689,E2 -11992.689} C_VEL
LIN {X 0,Y 383.002,Z 282.904,A -85,B 0,C 180,E1 -11996.128,E2 -11996.128} C_VEL
LIN {X 0,Y 383.528,Z 276.68,A -85,B 0,C 180,E1 -11999.653,E2 -11999.653} C_VEL
LIN {X 0,Y 384.198,Z 270.567,A -85,B 0,C 180,E1 -12003.282,E2 -12003.282} C_VEL
LIN {X 0,Y 384.416,Z 268.376,A -85,B 0,C 180,E1 -12004.642,E2 -12004.642} C_VEL
LIN {X 0,Y 384.314,Z 264.634,A -85,B 0,C 180,E1 -12007.118,E2 -12007.118} C_VEL
LIN {X 0,Y 383.84,Z 260.803,A -85,B 0,C 180,E1 -12009.853,E2 -12009.853} C_VEL
LIN {X 0,Y 383.094,Z 256.207,A -85,B 0,C 180,E1 -12013.466,E2 -12013.466} C_VEL
LIN {X 0,Y 383.021,Z 255.775,A -85,B 0,C 180,E1 -12013.84,E2 -12013.84} C_VEL
LIN {X 0,Y 383.039,Z 255.777,A -85,B 0,C 180,E1 -12017.243,E2 -12017.243} C_VEL
LIN {X 0,Y 383.02,Z 255.779,A -85,B 0,C 180,E1 -12020.411,E2 -12020.411} C_VEL
LIN {X 0,Y 383.025,Z 255.776,A -85,B 0,C 180,E1 -12024.043,E2 -12024.043} C_VEL
LIN {X 0,Y 382.986,Z 255.78,A -85,B 0,C 180,E1 -12027.576,E2 -12027.576} C_VEL
LIN {X 0,Y 382.995,Z 255.779,A -85,B 0,C 180,E1 -12030.299,E2 -12030.299} C_VEL
LIN {X 0,Y 383.053,Z 255.771,A -85,B 0,C 180,E1 -12032.697,E2 -12032.697} C_VEL
LIN {X 0,Y 383.029,Z 255.775,A -85,B 0,C 180,E1 -12036.191,E2 -12036.191} C_VEL
LIN {X 0,Y 383.051,Z 255.773,A -85,B 0,C 180,E1 -12039.597,E2 -12039.597} C_VEL
LIN {X 0,Y 383.1,Z 255.766,A -85,B 0,C 180,E1 -12042.93,E2 -12042.93} C_VEL
LIN {X 0,Y 383.12,Z 255.764,A -85,B 0,C 180,E1 -12046.463,E2 -12046.463} C_VEL
LIN {X 0,Y 383.146,Z 255.762,A -85,B 0,C 180,E1 -12050.497,E2 -12050.497} C_VEL
LIN {X 0,Y 383.267,Z 255.746,A -85,B 0,C 180,E1 -12052.624,E2 -12052.624} C_VEL
LIN {X 0,Y 383.193,Z 255.753,A -85,B 0,C 180,E1 -12054.737,E2 -12054.737} C_VEL
LIN {X 0,Y 383.381,Z 255.731,A -85,B 0,C 180,E1 -12057.898,E2 -12057.898} C_VEL
LIN {X 0,Y 383.511,Z 255.715,A -85,B 0,C 180,E1 -12059.999,E2 -12059.999} C_VEL
LIN {X 0,Y 383.246,Z 255.751,A -85,B 0,C 180,E1 -12063.152,E2 -12063.152} C_VEL
LIN {X 0,Y 383.255,Z 255.746,A -85,B 0,C 180,E1 -12066.636,E2 -12066.636} C_VEL
LIN {X 0,Y 383.251,Z 255.749,A -85,B 0,C 180,E1 -12067.374,E2 -12067.374} C_VEL
LIN {X 0,Y 383.326,Z 257.683,A -85,B 0,C 180,E1 -12069.496,E2 -12069.496} C_VEL
LIN {X 0,Y 383.25,Z 261.057,A -85,B 0,C 180,E1 -12072.711,E2 -12072.711} C_VEL
LIN {X 0,Y 382.948,Z 264.689,A -85,B 0,C 180,E1 -12075.978,E2 -12075.978} C_VEL
LIN {X 0,Y 382.766,Z 267.246,A -85,B 0,C 180,E1 -12078.187,E2 -12078.187} C_VEL
LIN {X 0,Y 382.454,Z 271.25,A -85,B 0,C 180,E1 -12081.561,E2 -12081.561} C_VEL
LIN {X 0,Y 382.216,Z 275.486,A -85,B 0,C 180,E1 -12085.017,E2 -12085.017} C_VEL
LIN {X 0,Y 382.104,Z 277.706,A -85,B 0,C 180,E1 -12086.782,E2 -12086.782} C_VEL
LIN {X 0,Y 385.695,Z 290.831,A -85,B 0,C 180,E1 -12087.5,E2 -12087.5} C_VEL
LIN {X 0,Y 388.25,Z 303.561,A -85,B 0,C 180,E1 -12088.358,E2 -12088.358} C_VEL
LIN {X 0,Y 388.322,Z 307.753,A -85,B 0,C 180,E1 -12088.65,E2 -12088.65} C_VEL
LIN {X 0,Y 387.5,Z 318.532,A -85,B 0,C 180,E1 -12089.478,E2 -12089.478} C_VEL
LIN {X 0,Y 386.499,Z 330.092,A -85,B 0,C 180,E1 -12090.605,E2 -12090.605} C_VEL
LIN {X 0,Y 385.436,Z 340.769,A -85,B 0,C 180,E1 -12091.921,E2 -12091.921} C_VEL
LIN {X 0,Y 384.535,Z 349.498,A -85,B 0,C 180,E1 -12093.248,E2 -12093.248} C_VEL
LIN {X 0,Y 383.732,Z 356.79,A -85,B 0,C 180,E1 -12094.592,E2 -12094.592} C_VEL
LIN {X 0,Y 382.938,Z 364.575,A -85,B 0,C 180,E1 -12096.384,E2 -12096.384} C_VEL
LIN {X 0,Y 382.344,Z 370.716,A -85,B 0,C 180,E1 -12098.207,E2 -12098.207} C_VEL
LIN {X 0,Y 381.887,Z 375.467,A -85,B 0,C 180,E1 -12100.097,E2 -12100.097} C_VEL
LIN {X 0,Y 381.671,Z 378.063,A -85,B 0,C 180,E1 -12101.519,E2 -12101.519} C_VEL
LIN {X 0,Y 381.543,Z 379.887,A -85,B 0,C 180,E1 -12102.962,E2 -12102.962} C_VEL
LIN {X 0,Y 381.436,Z 380.984,A -85,B 0,C 180,E1 -12104.437,E2 -12104.437} C_VEL
LIN {X 0,Y 381.392,Z 381.312,A -85,B 0,C 180,E1 -12105.942,E2 -12105.942} C_VEL
LIN {X 0,Y 381.362,Z 380.799,A -85,B 0,C 180,E1 -12107.486,E2 -12107.486} C_VEL
LIN {X 0,Y 381.484,Z 379.378,A -85,B 0,C 180,E1 -12109.052,E2 -12109.052} C_VEL
LIN {X 0,Y 381.64,Z 376.977,A -85,B 0,C 180,E1 -12110.661,E2 -12110.661} C_VEL
LIN {X 0,Y 381.962,Z 372.688,A -85,B 0,C 180,E1 -12112.614,E2 -12112.614} C_VEL
LIN {X 0,Y 382.387,Z 367.557,A -85,B 0,C 180,E1 -12114.319,E2 -12114.319} C_VEL
LIN {X 0,Y 382.934,Z 360.399,A -85,B 0,C 180,E1 -12116.16,E2 -12116.16} C_VEL
LIN {X 0,Y 383.668,Z 352.818,A -85,B 0,C 180,E1 -12117.693,E2 -12117.693} C_VEL
LIN {X 0,Y 384.44,Z 343.416,A -85,B 0,C 180,E1 -12119.225,E2 -12119.225} C_VEL
LIN {X 0,Y 385.224,Z 333.842,A -85,B 0,C 180,E1 -12120.49,E2 -12120.49} C_VEL
LIN {X 0,Y 386.089,Z 323.113,A -85,B 0,C 180,E1 -12121.63,E2 -12121.63} C_VEL
LIN {X 0,Y 386.844,Z 311.527,A -85,B 0,C 180,E1 -12122.609,E2 -12122.609} C_VEL
LIN {X 0,Y 387.369,Z 304.034,A -85,B 0,C 180,E1 -12123.123,E2 -12123.123} C_VEL
LIN {X 0,Y 385.15,Z 291.397,A -85,B 0,C 180,E1 -12123.919,E2 -12123.919} C_VEL
LIN {X 0,Y 382.227,Z 278.385,A -85,B 0,C 180,E1 -12124.553,E2 -12124.553} C_VEL
LIN {X 0,Y 381.938,Z 276.738,A -85,B 0,C 180,E1 -12124.656,E2 -12124.656} C_VEL
LIN {X 0,Y 382.145,Z 271.769,A -85,B 0,C 180,E1 -12128.419,E2 -12128.419} C_VEL
LIN {X 0,Y 382.288,Z 268.835,A -85,B 0,C 180,E1 -12130.676,E2 -12130.676} C_VEL
LIN {X 0,Y 382.477,Z 264.602,A -85,B 0,C 180,E1 -12134.001,E2 -12134.001} C_VEL
LIN {X 0,Y 382.753,Z 260.521,A -85,B 0,C 180,E1 -12137.271,E2 -12137.271} C_VEL
LIN {X 0,Y 382.927,Z 256.606,A -85,B 0,C 180,E1 -12140.493,E2 -12140.493} C_VEL
LIN {X 0,Y 383.021,Z 255.773,A -85,B 0,C 180,E1 -12141.559,E2 -12141.559} C_VEL
LIN {X 0,Y 383.245,Z 255.745,A -85,B 0,C 180,E1 -12143.683,E2 -12143.683} C_VEL
LIN {X 0,Y 383.377,Z 255.729,A -85,B 0,C 180,E1 -12147.899,E2 -12147.899} C_VEL
LIN {X 0,Y 383.511,Z 255.713,A -85,B 0,C 180,E1 -12150,E2 -12150} C_VEL
LIN {X 0,Y 383.242,Z 255.746,A -85,B 0,C 180,E1 -12153.154,E2 -12153.154} C_VEL
LIN {X 0,Y 383.277,Z 255.745,A -85,B 0,C 180,E1 -12156.316,E2 -12156.316} C_VEL
LIN {X 0,Y 383.25,Z 255.748,A -85,B 0,C 180,E1 -12158.436,E2 -12158.436} C_VEL
LIN {X 0,Y 383.097,Z 255.764,A -85,B 0,C 180,E1 -12161.642,E2 -12161.642} C_VEL
LIN {X 0,Y 383.104,Z 255.763,A -85,B 0,C 180,E1 -12164.882,E2 -12164.882} C_VEL
LIN {X 0,Y 383.083,Z 255.769,A -85,B 0,C 180,E1 -12168.172,E2 -12168.172} C_VEL
LIN {X 0,Y 383.057,Z 255.77,A -85,B 0,C 180,E1 -12170.332,E2 -12170.332} C_VEL
LIN {X 0,Y 382.421,Z 255.855,A -85,B 0,C 180,E1 -12171.21,E2 -12171.21} C_VEL
LIN {X 0,Y 379.544,Z 256.213,A -85,B 0,C 180,E1 -12172.636,E2 -12172.636} C_VEL
LIN {X 0,Y 377.093,Z 256.515,A -85,B 0,C 180,E1 -12173.79,E2 -12173.79} C_VEL
LIN {X 0,Y 376.051,Z 256.641,A -85,B 0,C 180,E1 -12174.682,E2 -12174.682} C_VEL
LIN {X 0,Y 375.973,Z 256.65,A -85,B 0,C 180,E1 -12174.985,E2 -12174.985} C_VEL
LIN {X 0,Y 375.992,Z 256.652,A -85,B 0,C 180,E1 -12177.859,E2 -12177.859} C_VEL
LIN {X 0,Y 375.965,Z 256.655,A -85,B 0,C 180,E1 -12181.561,E2 -12181.561} C_VEL
LIN {X 0,Y 375.948,Z 256.657,A -85,B 0,C 180,E1 -12185.416,E2 -12185.416} C_VEL
LIN {X 0,Y 375.967,Z 256.651,A -85,B 0,C 180,E1 -12188.272,E2 -12188.272} C_VEL
LIN {X 0,Y 375.979,Z 256.654,A -85,B 0,C 180,E1 -12191.611,E2 -12191.611} C_VEL
LIN {X 0,Y 376.005,Z 256.651,A -85,B 0,C 180,E1 -12195.256,E2 -12195.256} C_VEL
LIN {X 0,Y 375.99,Z 256.653,A -85,B 0,C 180,E1 -12199.142,E2 -12199.142} C_VEL
LIN {X 0,Y 375.958,Z 256.653,A -85,B 0,C 180,E1 -12201.913,E2 -12201.913} C_VEL
LIN {X 0,Y 375.97,Z 256.655,A -85,B 0,C 180,E1 -12205.334,E2 -12205.334} C_VEL
LIN {X 0,Y 375.95,Z 256.654,A -85,B 0,C 180,E1 -12208.439,E2 -12208.439} C_VEL
LIN {X 0,Y 375.993,Z 256.648,A -85,B 0,C 180,E1 -12212.143,E2 -12212.143} C_VEL
LIN {X 0,Y 375.997,Z 256.65,A -85,B 0,C 180,E1 -12214.54,E2 -12214.54} C_VEL
LIN {X 0,Y 375.954,Z 256.653,A -85,B 0,C 180,E1 -12218.047,E2 -12218.047} C_VEL
LIN {X 0,Y 376.001,Z 256.647,A -85,B 0,C 180,E1 -12221.474,E2 -12221.474} C_VEL
LIN {X 0,Y 376.05,Z 256.645,A -85,B 0,C 180,E1 -12224.834,E2 -12224.834} C_VEL
LIN {X 0,Y 376.043,Z 256.644,A -85,B 0,C 180,E1 -12228.138,E2 -12228.138} C_VEL
LIN {X 0,Y 376.213,Z 256.622,A -85,B 0,C 180,E1 -12231.92,E2 -12231.92} C_VEL
LIN {X 0,Y 376.164,Z 256.63,A -85,B 0,C 180,E1 -12234.641,E2 -12234.641} C_VEL
LIN {X 0,Y 376.348,Z 256.606,A -85,B 0,C 180,E1 -12237.861,E2 -12237.861} C_VEL
LIN {X 0,Y 376.483,Z 256.591,A -85,B 0,C 180,E1 -12240.001,E2 -12240.001} C_VEL
LIN {X 0,Y 376.185,Z 256.624,A -85,B 0,C 180,E1 -12243.214,E2 -12243.214} C_VEL
LIN {X 0,Y 376.241,Z 256.62,A -85,B 0,C 180,E1 -12246.436,E2 -12246.436} C_VEL
LIN {X 0,Y 376.202,Z 256.623,A -85,B 0,C 180,E1 -12248.596,E2 -12248.596} C_VEL
LIN {X 0,Y 376.055,Z 256.645,A -85,B 0,C 180,E1 -12251.864,E2 -12251.864} C_VEL
LIN {X 0,Y 376.056,Z 256.641,A -85,B 0,C 180,E1 -12255.169,E2 -12255.169} C_VEL
LIN {X 0,Y 376.006,Z 256.647,A -85,B 0,C 180,E1 -12258.528,E2 -12258.528} C_VEL
LIN {X 0,Y 375.96,Z 256.656,A -85,B 0,C 180,E1 -12261.956,E2 -12261.956} C_VEL
LIN {X 0,Y 376.005,Z 256.651,A -85,B 0,C 180,E1 -12265.462,E2 -12265.462} C_VEL
LIN {X 0,Y 375.959,Z 256.654,A -85,B 0,C 180,E1 -12269.081,E2 -12269.081} C_VEL
LIN {X 0,Y 375.948,Z 256.655,A -85,B 0,C 180,E1 -12272.83,E2 -12272.83} C_VEL
LIN {X 0,Y 375.957,Z 256.657,A -85,B 0,C 180,E1 -12275.417,E2 -12275.417} C_VEL
LIN {X 0,Y 375.975,Z 256.65,A -85,B 0,C 180,E1 -12278.272,E2 -12278.272} C_VEL
LIN {X 0,Y 375.935,Z 256.657,A -85,B 0,C 180,E1 -12281.602,E2 -12281.602} C_VEL
LIN {X 0,Y 375.928,Z 256.66,A -85,B 0,C 180,E1 -12285.27,E2 -12285.27} C_VEL
LIN {X 0,Y 375.978,Z 256.78,A -85,B 0,C 180,E1 -12288.393,E2 -12288.393} C_VEL
LIN {X 0,Y 376.842,Z 261.609,A -85,B 0,C 180,E1 -12291.564,E2 -12291.564} C_VEL
LIN {X 0,Y 377.223,Z 265.627,A -85,B 0,C 180,E1 -12294.065,E2 -12294.065} C_VEL
LIN {X 0,Y 377.162,Z 268.893,A -85,B 0,C 180,E1 -12296.013,E2 -12296.013} C_VEL
LIN {X 0,Y 376.485,Z 275.393,A -85,B 0,C 180,E1 -12299.734,E2 -12299.734} C_VEL
LIN {X 0,Y 375.927,Z 282.733,A -85,B 0,C 180,E1 -12303.816,E2 -12303.816} C_VEL
LIN {X 0,Y 375.449,Z 290.522,A -85,B 0,C 180,E1 -12308.014,E2 -12308.014} C_VEL
LIN {X 0,Y 375.124,Z 296.321,A -85,B 0,C 180,E1 -12311.074,E2 -12311.074} C_VEL
LIN {X 0,Y 377.568,Z 310.105,A -85,B 0,C 180,E1 -12311.681,E2 -12311.681} C_VEL
LIN {X 0,Y 379.353,Z 323.354,A -85,B 0,C 180,E1 -12312.472,E2 -12312.472} C_VEL
LIN {X 0,Y 379.909,Z 329.665,A -85,B 0,C 180,E1 -12312.922,E2 -12312.922} C_VEL
LIN {X 0,Y 378.993,Z 341.259,A -85,B 0,C 180,E1 -12313.85,E2 -12313.85} C_VEL
LIN {X 0,Y 378.067,Z 351.774,A -85,B 0,C 180,E1 -12314.915,E2 -12314.915} C_VEL
LIN {X 0,Y 377.174,Z 362.408,A -85,B 0,C 180,E1 -12316.257,E2 -12316.257} C_VEL
LIN {X 0,Y 376.441,Z 371.058,A -85,B 0,C 180,E1 -12317.602,E2 -12317.602} C_VEL
LIN {X 0,Y 375.629,Z 379.449,A -85,B 0,C 180,E1 -12319.216,E2 -12319.216} C_VEL
LIN {X 0,Y 375.152,Z 386.214,A -85,B 0,C 180,E1 -12320.837,E2 -12320.837} C_VEL
LIN {X 0,Y 374.785,Z 391.609,A -85,B 0,C 180,E1 -12322.457,E2 -12322.457} C_VEL
LIN {X 0,Y 374.59,Z 395.462,A -85,B 0,C 180,E1 -12323.928,E2 -12323.928} C_VEL
LIN {X 0,Y 374.552,Z 398.931,A -85,B 0,C 180,E1 -12325.696,E2 -12325.696} C_VEL
LIN {X 0,Y 374.464,Z 400.476,A -85,B 0,C 180,E1 -12326.772,E2 -12326.772} C_VEL
LIN {X 0,Y 374.463,Z 401.568,A -85,B 0,C 180,E1 -12327.849,E2 -12327.849} C_VEL
LIN {X 0,Y 374.519,Z 402.249,A -85,B 0,C 180,E1 -12328.925,E2 -12328.925} C_VEL
LIN {X 0,Y 374.555,Z 402.536,A -85,B 0,C 180,E1 -12330,E2 -12330} C_VEL
LIN {X 0,Y 374.504,Z 402.429,A -85,B 0,C 180,E1 -12331.075,E2 -12331.075} C_VEL
LIN {X 0,Y 374.459,Z 401.888,A -85,B 0,C 180,E1 -12332.151,E2 -12332.151} C_VEL
LIN {X 0,Y 374.53,Z 399.591,A -85,B 0,C 180,E1 -12334.304,E2 -12334.304} C_VEL
LIN {X 0,Y 374.569,Z 396.509,A -85,B 0,C 180,E1 -12336.042,E2 -12336.042} C_VEL
LIN {X 0,Y 374.806,Z 392.88,A -85,B 0,C 180,E1 -12337.542,E2 -12337.542} C_VEL
LIN {X 0,Y 375.199,Z 387.884,A -85,B 0,C 180,E1 -12339.161,E2 -12339.161} C_VEL
LIN {X 0,Y 375.796,Z 381.625,A -85,B 0,C 180,E1 -12340.778,E2 -12340.778} C_VEL
LIN {X 0,Y 376.611,Z 373.854,A -85,B 0,C 180,E1 -12342.392,E2 -12342.392} C_VEL
LIN {X 0,Y 377.635,Z 364.156,A -85,B 0,C 180,E1 -12344,E2 -12344} C_VEL
LIN {X 0,Y 378.554,Z 354.195,A -85,B 0,C 180,E1 -12345.34,E2 -12345.34} C_VEL
LIN {X 0,Y 379.723,Z 343.005,A -85,B 0,C 180,E1 -12346.532,E2 -12346.532} C_VEL
LIN {X 0,Y 380.83,Z 330.735,A -85,B 0,C 180,E1 -12347.564,E2 -12347.564} C_VEL
LIN {X 0,Y 379.854,Z 319.331,A -85,B 0,C 180,E1 -12348.402,E2 -12348.402} C_VEL
LIN {X 0,Y 377.801,Z 307.099,A -85,B 0,C 180,E1 -12349.148,E2 -12349.148} C_VEL
LIN {X 0,Y 375.232,Z 295.368,A -85,B 0,C 180,E1 -12349.755,E2 -12349.755} C_VEL
LIN {X 0,Y 375.601,Z 289.122,A -85,B 0,C 180,E1 -12353.137,E2 -12353.137} C_VEL
LIN {X 0,Y 376.037,Z 282.868,A -85,B 0,C 180,E1 -12356.65,E2 -12356.65} C_VEL
LIN {X 0,Y 376.578,Z 276.665,A -85,B 0,C 180,E1 -12360.257,E2 -12360.257} C_VEL
LIN {X 0,Y 377.321,Z 270.597,A -85,B 0,C 180,E1 -12363.971,E2 -12363.971} C_VEL
LIN {X 0,Y 377.358,Z 266.353,A -85,B 0,C 180,E1 -12366.788,E2 -12366.788} C_VEL
LIN {X 0,Y 376.967,Z 262.824,A -85,B 0,C 180,E1 -12369.336,E2 -12369.336} C_VEL
LIN {X 0,Y 376.396,Z 259.112,A -85,B 0,C 180,E1 -12372.235,E2 -12372.235} C_VEL
LIN {X 0,Y 375.954,Z 256.657,A -85,B 0,C 180,E1 -12374.481,E2 -12374.481} C_VEL
LIN {X 0,Y 375.96,Z 256.657,A -85,B 0,C 180,E1 -12377.702,E2 -12377.702} C_VEL
LIN {X 0,Y 375.968,Z 256.658,A -85,B 0,C 180,E1 -12380.537,E2 -12380.537} C_VEL
LIN {X 0,Y 375.964,Z 256.656,A -85,B 0,C 180,E1 -12383.494,E2 -12383.494} C_VEL
LIN {X 0,Y 375.958,Z 256.657,A -85,B 0,C 180,E1 -12385.887,E2 -12385.887} C_VEL
LIN {X 0,Y 375.965,Z 256.655,A -85,B 0,C 180,E1 -12389.686,E2 -12389.686} C_VEL
LIN {X 0,Y 375.999,Z 256.65,A -85,B 0,C 180,E1 -12392.14,E2 -12392.14} C_VEL
LIN {X 0,Y 376.003,Z 256.65,A -85,B 0,C 180,E1 -12394.538,E2 -12394.538} C_VEL
LIN {X 0,Y 375.959,Z 256.657,A -85,B 0,C 180,E1 -12398.044,E2 -12398.044} C_VEL
LIN {X 0,Y 376.004,Z 256.65,A -85,B 0,C 180,E1 -12401.472,E2 -12401.472} C_VEL
LIN {X 0,Y 376.053,Z 256.644,A -85,B 0,C 180,E1 -12404.831,E2 -12404.831} C_VEL
LIN {X 0,Y 376.045,Z 256.645,A -85,B 0,C 180,E1 -12408.135,E2 -12408.135} C_VEL
LIN {X 0,Y 376.251,Z 256.62,A -85,B 0,C 180,E1 -12411.876,E2 -12411.876} C_VEL
LIN {X 0,Y 376.165,Z 256.628,A -85,B 0,C 180,E1 -12414.639,E2 -12414.639} C_VEL
LIN {X 0,Y 376.347,Z 256.608,A -85,B 0,C 180,E1 -12417.858,E2 -12417.858} C_VEL
LIN {X 0,Y 376.481,Z 256.59,A -85,B 0,C 180,E1 -12419.999,E2 -12419.999} C_VEL
LIN {X 0,Y 376.184,Z 256.63,A -85,B 0,C 180,E1 -12423.212,E2 -12423.212} C_VEL
LIN {X 0,Y 376.227,Z 256.674,A -85,B 0,C 180,E1 -12426.632,E2 -12426.632} C_VEL
LIN {X 0,Y 376.25,Z 256.9,A -85,B 0,C 180,E1 -12427.512,E2 -12427.512} C_VEL
LIN {X 0,Y 376.32,Z 260.114,A -85,B 0,C 180,E1 -12430.762,E2 -12430.762} C_VEL
LIN {X 0,Y 376.092,Z 263.592,A -85,B 0,C 180,E1 -12434.058,E2 -12434.058} C_VEL
LIN {X 0,Y 375.832,Z 267.424,A -85,B 0,C 180,E1 -12437.509,E2 -12437.509} C_VEL
LIN {X 0,Y 375.484,Z 271.258,A -85,B 0,C 180,E1 -12440.83,E2 -12440.83} C_VEL
LIN {X 0,Y 375.2,Z 275.453,A -85,B 0,C 180,E1 -12444.334,E2 -12444.334} C_VEL
LIN {X 0,Y 375.094,Z 277.902,A -85,B 0,C 180,E1 -12446.332,E2 -12446.332} C_VEL
LIN {X 0,Y 379.121,Z 292.569,A -85,B 0,C 180,E1 -12447.196,E2 -12447.196} C_VEL
LIN {X 0,Y 381.454,Z 304.293,A -85,B 0,C 180,E1 -12448.021,E2 -12448.021} C_VEL
LIN {X 0,Y 381.632,Z 308.16,A -85,B 0,C 180,E1 -12448.306,E2 -12448.306} C_VEL
LIN {X 0,Y 380.798,Z 318.661,A -85,B 0,C 180,E1 -12449.127,E2 -12449.127} C_VEL
LIN {X 0,Y 379.862,Z 328.861,A -85,B 0,C 180,E1 -12450.121,E2 -12450.121} C_VEL
LIN {X 0,Y 378.776,Z 339.456,A -85,B 0,C 180,E1 -12451.407,E2 -12451.407} C_VEL
LIN {X 0,Y 377.72,Z 349.145,A -85,B 0,C 180,E1 -12452.875,E2 -12452.875} C_VEL
LIN {X 0,Y 376.763,Z 357.307,A -85,B 0,C 180,E1 -12454.4,E2 -12454.4} C_VEL
LIN {X 0,Y 375.923,Z 364.926,A -85,B 0,C 180,E1 -12456.203,E2 -12456.203} C_VEL
LIN {X 0,Y 375.287,Z 371.342,A -85,B 0,C 180,E1 -12458.167,E2 -12458.167} C_VEL
LIN {X 0,Y 374.872,Z 375.296,A -85,B 0,C 180,E1 -12459.768,E2 -12459.768} C_VEL
LIN {X 0,Y 374.596,Z 378.224,A -85,B 0,C 180,E1 -12461.371,E2 -12461.371} C_VEL
LIN {X 0,Y 374.449,Z 380.173,A -85,B 0,C 180,E1 -12462.948,E2 -12462.948} C_VEL
LIN {X 0,Y 374.335,Z 381.236,A -85,B 0,C 180,E1 -12464.486,E2 -12464.486} C_VEL
LIN {X 0,Y 374.29,Z 381.499,A -85,B 0,C 180,E1 -12465.994,E2 -12465.994} C_VEL
LIN {X 0,Y 374.267,Z 381.004,A -85,B 0,C 180,E1 -12467.469,E2 -12467.469} C_VEL
LIN {X 0,Y 374.375,Z 379.733,A -85,B 0,C 180,E1 -12468.927,E2 -12468.927} C_VEL
LIN {X 0,Y 374.606,Z 376.534,A -85,B 0,C 180,E1 -12471.062,E2 -12471.062} C_VEL
LIN {X 0,Y 374.861,Z 373.265,A -85,B 0,C 180,E1 -12472.555,E2 -12472.555} C_VEL
LIN {X 0,Y 375.35,Z 367.469,A -85,B 0,C 180,E1 -12474.52,E2 -12474.52} C_VEL
LIN {X 0,Y 375.871,Z 361.043,A -85,B 0,C 180,E1 -12476.204,E2 -12476.204} C_VEL
LIN {X 0,Y 376.679,Z 352.978,A -85,B 0,C 180,E1 -12477.877,E2 -12477.877} C_VEL
LIN {X 0,Y 377.391,Z 344.86,A -85,B 0,C 180,E1 -12479.242,E2 -12479.242} C_VEL
LIN {X 0,Y 378.237,Z 334.668,A -85,B 0,C 180,E1 -12480.64,E2 -12480.64} C_VEL
LIN {X 0,Y 379.104,Z 324.262,A -85,B 0,C 180,E1 -12481.789,E2 -12481.789} C_VEL
LIN {X 0,Y 379.946,Z 312.318,A -85,B 0,C 180,E1 -12482.829,E2 -12482.829} C_VEL
LIN {X 0,Y 380.429,Z 304.478,A -85,B 0,C 180,E1 -12483.386,E2 -12483.386} C_VEL
LIN {X 0,Y 378.194,Z 291.978,A -85,B 0,C 180,E1 -12484.2,E2 -12484.2} C_VEL
LIN {X 0,Y 375.121,Z 278.326,A -85,B 0,C 180,E1 -12484.884,E2 -12484.884} C_VEL
LIN {X 0,Y 374.86,Z 276.918,A -85,B 0,C 180,E1 -12484.976,E2 -12484.976} C_VEL
LIN {X 0,Y 375.054,Z 272.99,A -85,B 0,C 180,E1 -12487.99,E2 -12487.99} C_VEL
LIN {X 0,Y 375.232,Z 270.036,A -85,B 0,C 180,E1 -12490.298,E2 -12490.298} C_VEL
LIN {X 0,Y 375.418,Z 265.756,A -85,B 0,C 180,E1 -12493.692,E2 -12493.692} C_VEL
LIN {X 0,Y 375.679,Z 261.65,A -85,B 0,C 180,E1 -12497.028,E2 -12497.028} C_VEL
LIN {X 0,Y 375.856,Z 257.707,A -85,B 0,C 180,E1 -12500.312,E2 -12500.312} C_VEL
LIN {X 0,Y 375.954,Z 256.654,A -85,B 0,C 180,E1 -12501.399,E2 -12501.399} C_VEL
LIN {X 0,Y 376.197,Z 256.623,A -85,B 0,C 180,E1 -12503.564,E2 -12503.564} C_VEL
LIN {X 0,Y 376.344,Z 256.604,A -85,B 0,C 180,E1 -12507.86,E2 -12507.86} C_VEL
LIN {X 0,Y 376.48,Z 256.589,A -85,B 0,C 180,E1 -12510,E2 -12510} C_VEL
LIN {X 0,Y 376.181,Z 256.625,A -85,B 0,C 180,E1 -12513.213,E2 -12513.213} C_VEL
LIN {X 0,Y 376.236,Z 256.622,A -85,B 0,C 180,E1 -12516.435,E2 -12516.435} C_VEL
LIN {X 0,Y 376.196,Z 256.626,A -85,B 0,C 180,E1 -12518.595,E2 -12518.595} C_VEL
LIN {X 0,Y 376.049,Z 256.643,A -85,B 0,C 180,E1 -12521.863,E2 -12521.863} C_VEL
LIN {X 0,Y 376.052,Z 256.641,A -85,B 0,C 180,E1 -12525.168,E2 -12525.168} C_VEL
LIN {X 0,Y 376.02,Z 256.647,A -85,B 0,C 180,E1 -12528.526,E2 -12528.526} C_VEL
LIN {X 0,Y 375.969,Z 256.655,A -85,B 0,C 180,E1 -12531.954,E2 -12531.954} C_VEL
LIN {X 0,Y 375.973,Z 256.65,A -85,B 0,C 180,E1 -12534.985,E2 -12534.985} C_VEL
LIN {X 0,Y 375.331,Z 256.735,A -85,B 0,C 180,E1 -12535.878,E2 -12535.878} C_VEL
LIN {X 0,Y 372.501,Z 257.094,A -85,B 0,C 180,E1 -12537.332,E2 -12537.332} C_VEL
LIN {X 0,Y 370.075,Z 257.397,A -85,B 0,C 180,E1 -12538.507,E2 -12538.507} C_VEL
LIN {X 0,Y 369.01,Z 257.525,A -85,B 0,C 180,E1 -12539.416,E2 -12539.416} C_VEL
LIN {X 0,Y 368.911,Z 257.534,A -85,B 0,C 180,E1 -12539.724,E2 -12539.724} C_VEL
LIN {X 0,Y 368.889,Z 257.537,A -85,B 0,C 180,E1 -12543.538,E2 -12543.538} C_VEL
LIN {X 0,Y 368.893,Z 257.533,A -85,B 0,C 180,E1 -12546.857,E2 -12546.857} C_VEL
LIN {X 0,Y 368.942,Z 257.526,A -85,B 0,C 180,E1 -12550.365,E2 -12550.365} C_VEL
LIN {X 0,Y 368.964,Z 257.527,A -85,B 0,C 180,E1 -12553.632,E2 -12553.632} C_VEL
LIN {X 0,Y 368.94,Z 257.527,A -85,B 0,C 180,E1 -12556.706,E2 -12556.706} C_VEL
LIN {X 0,Y 368.943,Z 257.529,A -85,B 0,C 180,E1 -12559.636,E2 -12559.636} C_VEL
LIN {X 0,Y 368.894,Z 257.536,A -85,B 0,C 180,E1 -12563.145,E2 -12563.145} C_VEL
LIN {X 0,Y 368.887,Z 257.534,A -85,B 0,C 180,E1 -12566.463,E2 -12566.463} C_VEL
LIN {X 0,Y 368.914,Z 257.53,A -85,B 0,C 180,E1 -12570.311,E2 -12570.311} C_VEL
LIN {X 0,Y 368.973,Z 257.523,A -85,B 0,C 180,E1 -12573.536,E2 -12573.536} C_VEL
LIN {X 0,Y 368.958,Z 257.526,A -85,B 0,C 180,E1 -12576.423,E2 -12576.423} C_VEL
LIN {X 0,Y 368.928,Z 257.528,A -85,B 0,C 180,E1 -12579.948,E2 -12579.948} C_VEL
LIN {X 0,Y 368.967,Z 257.523,A -85,B 0,C 180,E1 -12583.4,E2 -12583.4} C_VEL
LIN {X 0,Y 369.05,Z 257.516,A -85,B 0,C 180,E1 -12586.791,E2 -12586.791} C_VEL
LIN {X 0,Y 369.061,Z 257.514,A -85,B 0,C 180,E1 -12590.133,E2 -12590.133} C_VEL
LIN {X 0,Y 369.194,Z 257.495,A -85,B 0,C 180,E1 -12593.443,E2 -12593.443} C_VEL
LIN {X 0,Y 369.313,Z 257.482,A -85,B 0,C 180,E1 -12597.82,E2 -12597.82} C_VEL
LIN {X 0,Y 369.452,Z 257.466,A -85,B 0,C 180,E1 -12600.001,E2 -12600.001} C_VEL
LIN {X 0,Y 369.314,Z 257.484,A -85,B 0,C 180,E1 -12602.182,E2 -12602.182} C_VEL
LIN {X 0,Y 369.203,Z 257.495,A -85,B 0,C 180,E1 -12606.56,E2 -12606.56} C_VEL
LIN {X 0,Y 369.135,Z 257.502,A -85,B 0,C 180,E1 -12608.762,E2 -12608.762} C_VEL
LIN {X 0,Y 369.009,Z 257.522,A -85,B 0,C 180,E1 -12612.094,E2 -12612.094} C_VEL
LIN {X 0,Y 368.995,Z 257.522,A -85,B 0,C 180,E1 -12615.466,E2 -12615.466} C_VEL
LIN {X 0,Y 368.955,Z 257.525,A -85,B 0,C 180,E1 -12618.895,E2 -12618.895} C_VEL
LIN {X 0,Y 368.93,Z 257.528,A -85,B 0,C 180,E1 -12622.396,E2 -12622.396} C_VEL
LIN {X 0,Y 368.998,Z 257.521,A -85,B 0,C 180,E1 -12625.981,E2 -12625.981} C_VEL
LIN {X 0,Y 368.913,Z 257.533,A -85,B 0,C 180,E1 -12629.692,E2 -12629.692} C_VEL
LIN {X 0,Y 368.896,Z 257.534,A -85,B 0,C 180,E1 -12633.044,E2 -12633.044} C_VEL
LIN {X 0,Y 368.917,Z 257.529,A -85,B 0,C 180,E1 -12636.198,E2 -12636.198} C_VEL
LIN {X 0,Y 368.905,Z 257.534,A -85,B 0,C 180,E1 -12638.954,E2 -12638.954} C_VEL
LIN {X 0,Y 368.882,Z 257.533,A -85,B 0,C 180,E1 -12642.01,E2 -12642.01} C_VEL
LIN {X 0,Y 368.881,Z 257.538,A -85,B 0,C 180,E1 -12645.177,E2 -12645.177} C_VEL
LIN {X 0,Y 368.947,Z 257.674,A -85,B 0,C 180,E1 -12648.187,E2 -12648.187} C_VEL
LIN {X 0,Y 369.717,Z 262.173,A -85,B 0,C 180,E1 -12651.205,E2 -12651.205} C_VEL
LIN {X 0,Y 370.212,Z 266.479,A -85,B 0,C 180,E1 -12653.95,E2 -12653.95} C_VEL
LIN {X 0,Y 369.985,Z 271.028,A -85,B 0,C 180,E1 -12656.7,E2 -12656.7} C_VEL
LIN {X 0,Y 369.352,Z 277.324,A -85,B 0,C 180,E1 -12660.349,E2 -12660.349} C_VEL
LIN {X 0,Y 368.837,Z 283.793,A -85,B 0,C 180,E1 -12664.008,E2 -12664.008} C_VEL
LIN {X 0,Y 368.341,Z 291.336,A -85,B 0,C 180,E1 -12668.157,E2 -12668.157} C_VEL
LIN {X 0,Y 368.078,Z 296.153,A -85,B 0,C 180,E1 -12670.752,E2 -12670.752} C_VEL
LIN {X 0,Y 370.446,Z 309.625,A -85,B 0,C 180,E1 -12671.346,E2 -12671.346} C_VEL
LIN {X 0,Y 372.183,Z 321.699,A -85,B 0,C 180,E1 -12672.075,E2 -12672.075} C_VEL
LIN {X 0,Y 372.97,Z 330.791,A -85,B 0,C 180,E1 -12672.736,E2 -12672.736} C_VEL
LIN {X 0,Y 372.01,Z 342.054,A -85,B 0,C 180,E1 -12673.679,E2 -12673.679} C_VEL
LIN {X 0,Y 371.028,Z 352.908,A -85,B 0,C 180,E1 -12674.824,E2 -12674.824} C_VEL
LIN {X 0,Y 370.244,Z 361.914,A -85,B 0,C 180,E1 -12675.994,E2 -12675.994} C_VEL
LIN {X 0,Y 369.485,Z 370.621,A -85,B 0,C 180,E1 -12677.365,E2 -12677.365} C_VEL
LIN {X 0,Y 368.605,Z 379.064,A -85,B 0,C 180,E1 -12679.008,E2 -12679.008} C_VEL
LIN {X 0,Y 368.087,Z 385.864,A -85,B 0,C 180,E1 -12680.66,E2 -12680.66} C_VEL
LIN {X 0,Y 367.714,Z 391.291,A -85,B 0,C 180,E1 -12682.311,E2 -12682.311} C_VEL
LIN {X 0,Y 367.508,Z 395.49,A -85,B 0,C 180,E1 -12683.95,E2 -12683.95} C_VEL
LIN {X 0,Y 367.458,Z 398.666,A -85,B 0,C 180,E1 -12685.612,E2 -12685.612} C_VEL
LIN {X 0,Y 367.382,Z 400.225,A -85,B 0,C 180,E1 -12686.71,E2 -12686.71} C_VEL
LIN {X 0,Y 367.363,Z 401.34,A -85,B 0,C 180,E1 -12687.807,E2 -12687.807} C_VEL
LIN {X 0,Y 367.419,Z 402.031,A -85,B 0,C 180,E1 -12688.904,E2 -12688.904} C_VEL
LIN {X 0,Y 367.458,Z 402.329,A -85,B 0,C 180,E1 -12690,E2 -12690} C_VEL
LIN {X 0,Y 367.404,Z 402.233,A -85,B 0,C 180,E1 -12691.096,E2 -12691.096} C_VEL
LIN {X 0,Y 367.36,Z 401.712,A -85,B 0,C 180,E1 -12692.193,E2 -12692.193} C_VEL
LIN {X 0,Y 367.379,Z 400.772,A -85,B 0,C 180,E1 -12693.29,E2 -12693.29} C_VEL
LIN {X 0,Y 367.438,Z 399.434,A -85,B 0,C 180,E1 -12694.388,E2 -12694.388} C_VEL
LIN {X 0,Y 367.478,Z 396.68,A -85,B 0,C 180,E1 -12696.006,E2 -12696.006} C_VEL
LIN {X 0,Y 367.733,Z 392.777,A -85,B 0,C 180,E1 -12697.688,E2 -12697.688} C_VEL
LIN {X 0,Y 368.164,Z 387.818,A -85,B 0,C 180,E1 -12699.338,E2 -12699.338} C_VEL
LIN {X 0,Y 368.766,Z 381.595,A -85,B 0,C 180,E1 -12700.986,E2 -12700.986} C_VEL
LIN {X 0,Y 369.676,Z 373.877,A -85,B 0,C 180,E1 -12702.628,E2 -12702.628} C_VEL
LIN {X 0,Y 370.721,Z 364.225,A -85,B 0,C 180,E1 -12704.267,E2 -12704.267} C_VEL
LIN {X 0,Y 371.697,Z 354.321,A -85,B 0,C 180,E1 -12705.63,E2 -12705.63} C_VEL
LIN {X 0,Y 372.942,Z 343.237,A -85,B 0,C 180,E1 -12706.842,E2 -12706.842} C_VEL
LIN {X 0,Y 374.05,Z 331.095,A -85,B 0,C 180,E1 -12707.891,E2 -12707.891} C_VEL
LIN {X 0,Y 372.937,Z 318.818,A -85,B 0,C 180,E1 -12708.827,E2 -12708.827} C_VEL
LIN {X 0,Y 370.713,Z 306.23,A -85,B 0,C 180,E1 -12709.621,E2 -12709.621} C_VEL
LIN {X 0,Y 368.201,Z 295.203,A -85,B 0,C 180,E1 -12710.187,E2 -12710.187} C_VEL
LIN {X 0,Y 368.539,Z 290.1,A -85,B 0,C 180,E1 -12713.012,E2 -12713.012} C_VEL
LIN {X 0,Y 368.944,Z 284.09,A -85,B 0,C 180,E1 -12716.451,E2 -12716.451} C_VEL
LIN {X 0,Y 369.549,Z 277.678,A -85,B 0,C 180,E1 -12720.262,E2 -12720.262} C_VEL
LIN {X 0,Y 370.167,Z 272.63,A -85,B 0,C 180,E1 -12723.407,E2 -12723.407} C_VEL
LIN {X 0,Y 370.39,Z 268.685,A -85,B 0,C 180,E1 -12726.029,E2 -12726.029} C_VEL
LIN {X 0,Y 370.081,Z 264.756,A -85,B 0,C 180,E1 -12728.865,E2 -12728.865} C_VEL
LIN {X 0,Y 369.477,Z 260.655,A -85,B 0,C 180,E1 -12732.111,E2 -12732.111} C_VEL
LIN {X 0,Y 368.891,Z 257.536,A -85,B 0,C 180,E1 -12734.912,E2 -12734.912} C_VEL
LIN {X 0,Y 368.909,Z 257.534,A -85,B 0,C 180,E1 -12738.18,E2 -12738.18} C_VEL
LIN {X 0,Y 368.912,Z 257.535,A -85,B 0,C 180,E1 -12741.357,E2 -12741.357} C_VEL
LIN {X 0,Y 368.935,Z 257.53,A -85,B 0,C 180,E1 -12745.145,E2 -12745.145} C_VEL
LIN {X 0,Y 368.927,Z 257.532,A -85,B 0,C 180,E1 -12749.045,E2 -12749.045} C_VEL
LIN {X 0,Y 368.984,Z 257.524,A -85,B 0,C 180,E1 -12751.563,E2 -12751.563} C_VEL
LIN {X 0,Y 368.954,Z 257.528,A -85,B 0,C 180,E1 -12755.223,E2 -12755.223} C_VEL
LIN {X 0,Y 368.933,Z 257.531,A -85,B 0,C 180,E1 -12758.972,E2 -12758.972} C_VEL
LIN {X 0,Y 368.986,Z 257.524,A -85,B 0,C 180,E1 -12762.256,E2 -12762.256} C_VEL
LIN {X 0,Y 369.032,Z 257.519,A -85,B 0,C 180,E1 -12766.226,E2 -12766.226} C_VEL
LIN {X 0,Y 369.062,Z 257.515,A -85,B 0,C 180,E1 -12770.13,E2 -12770.13} C_VEL
LIN {X 0,Y 369.182,Z 257.5,A -85,B 0,C 180,E1 -12772.341,E2 -12772.341} C_VEL
LIN {X 0,Y 369.138,Z 257.504,A -85,B 0,C 180,E1 -12774.536,E2 -12774.536} C_VEL
LIN {X 0,Y 369.312,Z 257.484,A -85,B 0,C 180,E1 -12777.818,E2 -12777.818} C_VEL
LIN {X 0,Y 369.45,Z 257.466,A -85,B 0,C 180,E1 -12779.999,E2 -12779.999} C_VEL
LIN {X 0,Y 369.311,Z 257.485,A -85,B 0,C 180,E1 -12782.18,E2 -12782.18} C_VEL
LIN {X 0,Y 369.201,Z 257.551,A -85,B 0,C 180,E1 -12786.635,E2 -12786.635} C_VEL
LIN {X 0,Y 369.314,Z 259.269,A -85,B 0,C 180,E1 -12788.755,E2 -12788.755} C_VEL
LIN {X 0,Y 369.24,Z 262.587,A -85,B 0,C 180,E1 -12792.084,E2 -12792.084} C_VEL
LIN {X 0,Y 368.929,Z 266.166,A -85,B 0,C 180,E1 -12795.466,E2 -12795.466} C_VEL
LIN {X 0,Y 368.754,Z 268.677,A -85,B 0,C 180,E1 -12797.753,E2 -12797.753} C_VEL
LIN {X 0,Y 368.387,Z 272.66,A -85,B 0,C 180,E1 -12801.251,E2 -12801.251} C_VEL
LIN {X 0,Y 368.102,Z 276.881,A -85,B 0,C 180,E1 -12804.835,E2 -12804.835} C_VEL
LIN {X 0,Y 368.11,Z 278.246,A -85,B 0,C 180,E1 -12805.894,E2 -12805.894} C_VEL
LIN {X 0,Y 371.832,Z 291.423,A -85,B 0,C 180,E1 -12806.677,E2 -12806.677} C_VEL
LIN {X 0,Y 374.363,Z 303.32,A -85,B 0,C 180,E1 -12807.533,E2 -12807.533} C_VEL
LIN {X 0,Y 374.981,Z 308.46,A -85,B 0,C 180,E1 -12807.939,E2 -12807.939} C_VEL
LIN {X 0,Y 373.925,Z 320.813,A -85,B 0,C 180,E1 -12808.943,E2 -12808.943} C_VEL
LIN {X 0,Y 372.856,Z 331.609,A -85,B 0,C 180,E1 -12810.071,E2 -12810.071} C_VEL
LIN {X 0,Y 371.794,Z 341.293,A -85,B 0,C 180,E1 -12811.319,E2 -12811.319} C_VEL
LIN {X 0,Y 370.77,Z 350.033,A -85,B 0,C 180,E1 -12812.697,E2 -12812.697} C_VEL
LIN {X 0,Y 369.875,Z 357.301,A -85,B 0,C 180,E1 -12814.091,E2 -12814.091} C_VEL
LIN {X 0,Y 368.968,Z 364.887,A -85,B 0,C 180,E1 -12815.902,E2 -12815.902} C_VEL
LIN {X 0,Y 368.375,Z 370.543,A -85,B 0,C 180,E1 -12817.624,E2 -12817.624} C_VEL
LIN {X 0,Y 367.842,Z 375.492,A -85,B 0,C 180,E1 -12819.6,E2 -12819.6} C_VEL
LIN {X 0,Y 367.635,Z 377.3,A -85,B 0,C 180,E1 -12820.537,E2 -12820.537} C_VEL
LIN {X 0,Y 367.435,Z 379.486,A -85,B 0,C 180,E1 -12822.022,E2 -12822.022} C_VEL
LIN {X 0,Y 367.306,Z 380.94,A -85,B 0,C 180,E1 -12823.535,E2 -12823.535} C_VEL
LIN {X 0,Y 367.209,Z 381.653,A -85,B 0,C 180,E1 -12825.082,E2 -12825.082} C_VEL
LIN {X 0,Y 367.161,Z 381.57,A -85,B 0,C 180,E1 -12826.664,E2 -12826.664} C_VEL
LIN {X 0,Y 367.233,Z 380.604,A -85,B 0,C 180,E1 -12828.274,E2 -12828.274} C_VEL
LIN {X 0,Y 367.364,Z 378.7,A -85,B 0,C 180,E1 -12829.925,E2 -12829.925} C_VEL
LIN {X 0,Y 367.632,Z 375.773,A -85,B 0,C 180,E1 -12831.606,E2 -12831.606} C_VEL
LIN {X 0,Y 367.938,Z 371.63,A -85,B 0,C 180,E1 -12833.342,E2 -12833.342} C_VEL
LIN {X 0,Y 368.398,Z 366.069,A -85,B 0,C 180,E1 -12835.114,E2 -12835.114} C_VEL
LIN {X 0,Y 369.105,Z 358.837,A -85,B 0,C 180,E1 -12836.904,E2 -12836.904} C_VEL
LIN {X 0,Y 369.898,Z 350.403,A -85,B 0,C 180,E1 -12838.572,E2 -12838.572} C_VEL
LIN {X 0,Y 370.747,Z 341.387,A -85,B 0,C 180,E1 -12840.003,E2 -12840.003} C_VEL
LIN {X 0,Y 371.645,Z 331.106,A -85,B 0,C 180,E1 -12841.325,E2 -12841.325} C_VEL
LIN {X 0,Y 372.574,Z 320.31,A -85,B 0,C 180,E1 -12842.442,E2 -12842.442} C_VEL
LIN {X 0,Y 373.367,Z 308.995,A -85,B 0,C 180,E1 -12843.371,E2 -12843.371} C_VEL
LIN {X 0,Y 373.544,Z 305.564,A -85,B 0,C 180,E1 -12843.61,E2 -12843.61} C_VEL
LIN {X 0,Y 371.323,Z 293.098,A -85,B 0,C 180,E1 -12844.458,E2 -12844.458} C_VEL
LIN {X 0,Y 368.402,Z 279.801,A -85,B 0,C 180,E1 -12845.148,E2 -12845.148} C_VEL
LIN {X 0,Y 367.816,Z 277.122,A -85,B 0,C 180,E1 -12845.294,E2 -12845.294} C_VEL
LIN {X 0,Y 368.103,Z 271.984,A -85,B 0,C 180,E1 -12849.309,E2 -12849.309} C_VEL
LIN {X 0,Y 368.339,Z 266.922,A -85,B 0,C 180,E1 -12853.37,E2 -12853.37} C_VEL
LIN {X 0,Y 368.601,Z 262.785,A -85,B 0,C 180,E1 -12856.774,E2 -12856.774} C_VEL
LIN {X 0,Y 368.804,Z 258.817,A -85,B 0,C 180,E1 -12860.125,E2 -12860.125} C_VEL
LIN {X 0,Y 368.888,Z 257.535,A -85,B 0,C 180,E1 -12861.233,E2 -12861.233} C_VEL
LIN {X 0,Y 369.149,Z 257.501,A -85,B 0,C 180,E1 -12863.441,E2 -12863.441} C_VEL
LIN {X 0,Y 369.309,Z 257.48,A -85,B 0,C 180,E1 -12867.819,E2 -12867.819} C_VEL
LIN {X 0,Y 369.45,Z 257.464,A -85,B 0,C 180,E1 -12870,E2 -12870} C_VEL
LIN {X 0,Y 369.309,Z 257.483,A -85,B 0,C 180,E1 -12872.181,E2 -12872.181} C_VEL
LIN {X 0,Y 369.198,Z 257.498,A -85,B 0,C 180,E1 -12876.558,E2 -12876.558} C_VEL
LIN {X 0,Y 369.128,Z 257.505,A -85,B 0,C 180,E1 -12878.761,E2 -12878.761} C_VEL
LIN {X 0,Y 369.003,Z 257.523,A -85,B 0,C 180,E1 -12882.093,E2 -12882.093} C_VEL
LIN {X 0,Y 368.991,Z 257.521,A -85,B 0,C 180,E1 -12885.465,E2 -12885.465} C_VEL
LIN {X 0,Y 368.98,Z 257.522,A -85,B 0,C 180,E1 -12888.893,E2 -12888.893} C_VEL
LIN {X 0,Y 368.936,Z 257.529,A -85,B 0,C 180,E1 -12892.395,E2 -12892.395} C_VEL
LIN {X 0,Y 368.989,Z 257.525,A -85,B 0,C 180,E1 -12895.981,E2 -12895.981} C_VEL
LIN {X 0,Y 368.957,Z 257.524,A -85,B 0,C 180,E1 -12898.814,E2 -12898.814} C_VEL
LIN {X 0,Y 368.911,Z 257.534,A -85,B 0,C 180,E1 -12899.724,E2 -12899.724} C_VEL
LIN {X 0,Y 368.211,Z 257.618,A -85,B 0,C 180,E1 -12900.635,E2 -12900.635} C_VEL
LIN {X 0,Y 365.351,Z 257.975,A -85,B 0,C 180,E1 -12902.117,E2 -12902.117} C_VEL
LIN {X 0,Y 362.949,Z 258.275,A -85,B 0,C 180,E1 -12903.315,E2 -12903.315} C_VEL
LIN {X 0,Y 361.921,Z 258.402,A -85,B 0,C 180,E1 -12904.242,E2 -12904.242} C_VEL
LIN {X 0,Y 361.838,Z 258.411,A -85,B 0,C 180,E1 -12904.556,E2 -12904.556} C_VEL
LIN {X 0,Y 361.864,Z 258.407,A -85,B 0,C 180,E1 -12908.425,E2 -12908.425} C_VEL
LIN {X 0,Y 361.864,Z 258.412,A -85,B 0,C 180,E1 -12911.325,E2 -12911.325} C_VEL
LIN {X 0,Y 361.923,Z 258.4,A -85,B 0,C 180,E1 -12914.351,E2 -12914.351} C_VEL
LIN {X 0,Y 361.876,Z 258.409,A -85,B 0,C 180,E1 -12917.56,E2 -12917.56} C_VEL
LIN {X 0,Y 361.866,Z 258.411,A -85,B 0,C 180,E1 -12920.973,E2 -12920.973} C_VEL
LIN {X 0,Y 361.865,Z 258.409,A -85,B 0,C 180,E1 -12924.656,E2 -12924.656} C_VEL
LIN {X 0,Y 361.829,Z 258.412,A -85,B 0,C 180,E1 -12928.372,E2 -12928.372} C_VEL
LIN {X 0,Y 361.894,Z 258.409,A -85,B 0,C 180,E1 -12930.956,E2 -12930.956} C_VEL
LIN {X 0,Y 361.946,Z 258.398,A -85,B 0,C 180,E1 -12933.476,E2 -12933.476} C_VEL
LIN {X 0,Y 361.881,Z 258.408,A -85,B 0,C 180,E1 -12937.146,E2 -12937.146} C_VEL
LIN {X 0,Y 361.898,Z 258.408,A -85,B 0,C 180,E1 -12940.725,E2 -12940.725} C_VEL
LIN {X 0,Y 361.925,Z 258.402,A -85,B 0,C 180,E1 -12943.067,E2 -12943.067} C_VEL
LIN {X 0,Y 361.992,Z 258.397,A -85,B 0,C 180,E1 -12946.529,E2 -12946.529} C_VEL
LIN {X 0,Y 362.025,Z 258.388,A -85,B 0,C 180,E1 -12949.939,E2 -12949.939} C_VEL
LIN {X 0,Y 362.156,Z 258.371,A -85,B 0,C 180,E1 -12953.315,E2 -12953.315} C_VEL
LIN {X 0,Y 362.277,Z 258.358,A -85,B 0,C 180,E1 -12957.778,E2 -12957.778} C_VEL
LIN {X 0,Y 362.422,Z 258.342,A -85,B 0,C 180,E1 -12960.001,E2 -12960.001} C_VEL
LIN {X 0,Y 362.278,Z 258.361,A -85,B 0,C 180,E1 -12962.225,E2 -12962.225} C_VEL
LIN {X 0,Y 362.167,Z 258.371,A -85,B 0,C 180,E1 -12966.688,E2 -12966.688} C_VEL
LIN {X 0,Y 362.071,Z 258.382,A -85,B 0,C 180,E1 -12968.935,E2 -12968.935} C_VEL
LIN {X 0,Y 361.963,Z 258.398,A -85,B 0,C 180,E1 -12972.333,E2 -12972.333} C_VEL
LIN {X 0,Y 361.959,Z 258.396,A -85,B 0,C 180,E1 -12974.622,E2 -12974.622} C_VEL
LIN {X 0,Y 361.953,Z 258.399,A -85,B 0,C 180,E1 -12978.101,E2 -12978.101} C_VEL
LIN {X 0,Y 361.89,Z 258.409,A -85,B 0,C 180,E1 -12981.654,E2 -12981.654} C_VEL
LIN {X 0,Y 361.927,Z 258.403,A -85,B 0,C 180,E1 -12985.291,E2 -12985.291} C_VEL
LIN {X 0,Y 361.907,Z 258.406,A -85,B 0,C 180,E1 -12987.78,E2 -12987.78} C_VEL
LIN {X 0,Y 361.837,Z 258.415,A -85,B 0,C 180,E1 -12991.631,E2 -12991.631} C_VEL
LIN {X 0,Y 361.874,Z 258.411,A -85,B 0,C 180,E1 -12995.346,E2 -12995.346} C_VEL
LIN {X 0,Y 361.871,Z 258.41,A -85,B 0,C 180,E1 -12999.028,E2 -12999.028} C_VEL
LIN {X 0,Y 361.837,Z 258.414,A -85,B 0,C 180,E1 -13002.83,E2 -13002.83} C_VEL
LIN {X 0,Y 361.819,Z 258.416,A -85,B 0,C 180,E1 -13005.948,E2 -13005.948} C_VEL
LIN {X 0,Y 361.908,Z 258.575,A -85,B 0,C 180,E1 -13007.991,E2 -13007.991} C_VEL
LIN {X 0,Y 362.62,Z 262.716,A -85,B 0,C 180,E1 -13010.829,E2 -13010.829} C_VEL
LIN {X 0,Y 363.082,Z 266.21,A -85,B 0,C 180,E1 -13013.127,E2 -13013.127} C_VEL
LIN {X 0,Y 363.15,Z 269.482,A -85,B 0,C 180,E1 -13015.187,E2 -13015.187} C_VEL
LIN {X 0,Y 362.625,Z 275.013,A -85,B 0,C 180,E1 -13018.515,E2 -13018.515} C_VEL
LIN {X 0,Y 361.932,Z 281.377,A -85,B 0,C 180,E1 -13022.223,E2 -13022.223} C_VEL
LIN {X 0,Y 361.58,Z 286.775,A -85,B 0,C 180,E1 -13025.299,E2 -13025.299} C_VEL
LIN {X 0,Y 361.176,Z 293.525,A -85,B 0,C 180,E1 -13029.072,E2 -13029.072} C_VEL
LIN {X 0,Y 361.026,Z 295.96,A -85,B 0,C 180,E1 -13030.416,E2 -13030.416} C_VEL
LIN {X 0,Y 363.392,Z 309.571,A -85,B 0,C 180,E1 -13031.034,E2 -13031.034} C_VEL
LIN {X 0,Y 365.185,Z 321.679,A -85,B 0,C 180,E1 -13031.783,E2 -13031.783} C_VEL
LIN {X 0,Y 366.038,Z 331.759,A -85,B 0,C 180,E1 -13032.542,E2 -13032.542} C_VEL
LIN {X 0,Y 364.921,Z 344.217,A -85,B 0,C 180,E1 -13033.641,E2 -13033.641} C_VEL
LIN {X 0,Y 363.939,Z 354.521,A -85,B 0,C 180,E1 -13034.794,E2 -13034.794} C_VEL
LIN {X 0,Y 362.956,Z 365.095,A -85,B 0,C 180,E1 -13036.279,E2 -13036.279} C_VEL
LIN {X 0,Y 362.168,Z 373.193,A -85,B 0,C 180,E1 -13037.675,E2 -13037.675} C_VEL
LIN {X 0,Y 361.414,Z 381.142,A -85,B 0,C 180,E1 -13039.354,E2 -13039.354} C_VEL
LIN {X 0,Y 360.916,Z 387.483,A -85,B 0,C 180,E1 -13041.038,E2 -13041.038} C_VEL
LIN {X 0,Y 360.592,Z 392.52,A -85,B 0,C 180,E1 -13042.722,E2 -13042.722} C_VEL
LIN {X 0,Y 360.387,Z 396.403,A -85,B 0,C 180,E1 -13044.404,E2 -13044.404} C_VEL
LIN {X 0,Y 360.367,Z 398.399,A -85,B 0,C 180,E1 -13045.526,E2 -13045.526} C_VEL
LIN {X 0,Y 360.302,Z 399.97,A -85,B 0,C 180,E1 -13046.645,E2 -13046.645} C_VEL
LIN {X 0,Y 360.268,Z 401.109,A -85,B 0,C 180,E1 -13047.764,E2 -13047.764} C_VEL
LIN {X 0,Y 360.319,Z 401.811,A -85,B 0,C 180,E1 -13048.882,E2 -13048.882} C_VEL
LIN {X 0,Y 360.361,Z 402.121,A -85,B 0,C 180,E1 -13050,E2 -13050} C_VEL
LIN {X 0,Y 360.304,Z 402.037,A -85,B 0,C 180,E1 -13051.117,E2 -13051.117} C_VEL
LIN {X 0,Y 360.264,Z 401.541,A -85,B 0,C 180,E1 -13052.236,E2 -13052.236} C_VEL
LIN {X 0,Y 360.299,Z 400.614,A -85,B 0,C 180,E1 -13053.355,E2 -13053.355} C_VEL
LIN {X 0,Y 360.349,Z 399.29,A -85,B 0,C 180,E1 -13054.474,E2 -13054.474} C_VEL
LIN {X 0,Y 360.381,Z 396.881,A -85,B 0,C 180,E1 -13055.961,E2 -13055.961} C_VEL
LIN {X 0,Y 360.683,Z 392.688,A -85,B 0,C 180,E1 -13057.839,E2 -13057.839} C_VEL
LIN {X 0,Y 361.118,Z 387.756,A -85,B 0,C 180,E1 -13059.522,E2 -13059.522} C_VEL
LIN {X 0,Y 361.753,Z 381.564,A -85,B 0,C 180,E1 -13061.202,E2 -13061.202} C_VEL
LIN {X 0,Y 362.749,Z 373.893,A -85,B 0,C 180,E1 -13062.873,E2 -13062.873} C_VEL
LIN {X 0,Y 363.667,Z 366.074,A -85,B 0,C 180,E1 -13064.264,E2 -13064.264} C_VEL
LIN {X 0,Y 364.64,Z 356.598,A -85,B 0,C 180,E1 -13065.654,E2 -13065.654} C_VEL
LIN {X 0,Y 365.831,Z 346.169,A -85,B 0,C 180,E1 -13066.891,E2 -13066.891} C_VEL
LIN {X 0,Y 367.131,Z 334.768,A -85,B 0,C 180,E1 -13067.969,E2 -13067.969} C_VEL
LIN {X 0,Y 367.078,Z 328.301,A -85,B 0,C 180,E1 -13068.51,E2 -13068.51} C_VEL
LIN {X 0,Y 365.825,Z 317.216,A -85,B 0,C 180,E1 -13069.353,E2 -13069.353} C_VEL
LIN {X 0,Y 363.584,Z 305.125,A -85,B 0,C 180,E1 -13070.127,E2 -13070.127} C_VEL
LIN {X 0,Y 361.175,Z 294.984,A -85,B 0,C 180,E1 -13070.668,E2 -13070.668} C_VEL
LIN {X 0,Y 361.581,Z 288.991,A -85,B 0,C 180,E1 -13074.089,E2 -13074.089} C_VEL
LIN {X 0,Y 362.112,Z 282.769,A -85,B 0,C 180,E1 -13077.761,E2 -13077.761} C_VEL
LIN {X 0,Y 362.766,Z 276.677,A -85,B 0,C 180,E1 -13081.538,E2 -13081.538} C_VEL
LIN {X 0,Y 363.237,Z 272.684,A -85,B 0,C 180,E1 -13084.131,E2 -13084.131} C_VEL
LIN {X 0,Y 363.406,Z 270.391,A -85,B 0,C 180,E1 -13085.682,E2 -13085.682} C_VEL
LIN {X 0,Y 363.186,Z 266.856,A -85,B 0,C 180,E1 -13088.259,E2 -13088.259} C_VEL
LIN {X 0,Y 362.657,Z 263.121,A -85,B 0,C 180,E1 -13091.214,E2 -13091.214} C_VEL
LIN {X 0,Y 362.078,Z 259.557,A -85,B 0,C 180,E1 -13094.327,E2 -13094.327} C_VEL
LIN {X 0,Y 361.822,Z 258.418,A -85,B 0,C 180,E1 -13095.631,E2 -13095.631} C_VEL
LIN {X 0,Y 361.872,Z 258.414,A -85,B 0,C 180,E1 -13099.236,E2 -13099.236} C_VEL
LIN {X 0,Y 361.868,Z 258.411,A -85,B 0,C 180,E1 -13102.981,E2 -13102.981} C_VEL
LIN {X 0,Y 361.857,Z 258.412,A -85,B 0,C 180,E1 -13106.629,E2 -13106.629} C_VEL
LIN {X 0,Y 361.874,Z 258.41,A -85,B 0,C 180,E1 -13109.671,E2 -13109.671} C_VEL
LIN {X 0,Y 361.951,Z 258.4,A -85,B 0,C 180,E1 -13113.474,E2 -13113.474} C_VEL
LIN {X 0,Y 361.886,Z 258.408,A -85,B 0,C 180,E1 -13117.143,E2 -13117.143} C_VEL
LIN {X 0,Y 361.902,Z 258.407,A -85,B 0,C 180,E1 -13120.722,E2 -13120.722} C_VEL
LIN {X 0,Y 361.928,Z 258.404,A -85,B 0,C 180,E1 -13123.065,E2 -13123.065} C_VEL
LIN {X 0,Y 361.993,Z 258.395,A -85,B 0,C 180,E1 -13126.526,E2 -13126.526} C_VEL
LIN {X 0,Y 362.026,Z 258.391,A -85,B 0,C 180,E1 -13129.937,E2 -13129.937} C_VEL
LIN {X 0,Y 362.145,Z 258.377,A -85,B 0,C 180,E1 -13132.191,E2 -13132.191} C_VEL
LIN {X 0,Y 362.112,Z 258.379,A -85,B 0,C 180,E1 -13134.43,E2 -13134.43} C_VEL
LIN {X 0,Y 362.276,Z 258.36,A -85,B 0,C 180,E1 -13137.775,E2 -13137.775} C_VEL
LIN {X 0,Y 362.42,Z 258.342,A -85,B 0,C 180,E1 -13139.999,E2 -13139.999} C_VEL
LIN {X 0,Y 362.275,Z 258.362,A -85,B 0,C 180,E1 -13142.222,E2 -13142.222} C_VEL
LIN {X 0,Y 362.175,Z 258.597,A -85,B 0,C 180,E1 -13146.685,E2 -13146.685} C_VEL
LIN {X 0,Y 362.312,Z 260.624,A -85,B 0,C 180,E1 -13148.926,E2 -13148.926} C_VEL
LIN {X 0,Y 362.19,Z 263.934,A -85,B 0,C 180,E1 -13152.323,E2 -13152.323} C_VEL
LIN {X 0,Y 361.881,Z 267.532,A -85,B 0,C 180,E1 -13155.775,E2 -13155.775} C_VEL
LIN {X 0,Y 361.52,Z 271.361,A -85,B 0,C 180,E1 -13159.296,E2 -13159.296} C_VEL
LIN {X 0,Y 361.198,Z 275.455,A -85,B 0,C 180,E1 -13162.9,E2 -13162.9} C_VEL
LIN {X 0,Y 361.083,Z 278.355,A -85,B 0,C 180,E1 -13165.39,E2 -13165.39} C_VEL
LIN {X 0,Y 365.525,Z 294.149,A -85,B 0,C 180,E1 -13166.403,E2 -13166.403} C_VEL
LIN {X 0,Y 367.882,Z 305.718,A -85,B 0,C 180,E1 -13167.288,E2 -13167.288} C_VEL
LIN {X 0,Y 368.224,Z 310.615,A -85,B 0,C 180,E1 -13167.685,E2 -13167.685} C_VEL
LIN {X 0,Y 367.026,Z 322.973,A -85,B 0,C 180,E1 -13168.756,E2 -13168.756} C_VEL
LIN {X 0,Y 365.858,Z 333.898,A -85,B 0,C 180,E1 -13169.962,E2 -13169.962} C_VEL
LIN {X 0,Y 364.661,Z 343.977,A -85,B 0,C 180,E1 -13171.355,E2 -13171.355} C_VEL
LIN {X 0,Y 363.511,Z 353.408,A -85,B 0,C 180,E1 -13172.983,E2 -13172.983} C_VEL
LIN {X 0,Y 362.56,Z 360.51,A -85,B 0,C 180,E1 -13174.49,E2 -13174.49} C_VEL
LIN {X 0,Y 361.729,Z 367.462,A -85,B 0,C 180,E1 -13176.338,E2 -13176.338} C_VEL
LIN {X 0,Y 361.243,Z 371.826,A -85,B 0,C 180,E1 -13177.792,E2 -13177.792} C_VEL
LIN {X 0,Y 360.801,Z 375.616,A -85,B 0,C 180,E1 -13179.389,E2 -13179.389} C_VEL
LIN {X 0,Y 360.407,Z 379.222,A -85,B 0,C 180,E1 -13181.527,E2 -13181.527} C_VEL
LIN {X 0,Y 360.182,Z 381.386,A -85,B 0,C 180,E1 -13183.785,E2 -13183.785} C_VEL
LIN {X 0,Y 360.098,Z 381.9,A -85,B 0,C 180,E1 -13185.365,E2 -13185.365} C_VEL
LIN {X 0,Y 360.072,Z 381.647,A -85,B 0,C 180,E1 -13186.912,E2 -13186.912} C_VEL
LIN {X 0,Y 360.139,Z 380.668,A -85,B 0,C 180,E1 -13188.434,E2 -13188.434} C_VEL
LIN {X 0,Y 360.365,Z 377.862,A -85,B 0,C 180,E1 -13190.629,E2 -13190.629} C_VEL
LIN {X 0,Y 360.611,Z 375.004,A -85,B 0,C 180,E1 -13192.129,E2 -13192.129} C_VEL
LIN {X 0,Y 360.959,Z 371.266,A -85,B 0,C 180,E1 -13193.642,E2 -13193.642} C_VEL
LIN {X 0,Y 361.528,Z 364.657,A -85,B 0,C 180,E1 -13195.685,E2 -13195.685} C_VEL
LIN {X 0,Y 362.203,Z 357.454,A -85,B 0,C 180,E1 -13197.423,E2 -13197.423} C_VEL
LIN {X 0,Y 362.942,Z 350.358,A -85,B 0,C 180,E1 -13198.81,E2 -13198.81} C_VEL
LIN {X 0,Y 363.867,Z 340.643,A -85,B 0,C 180,E1 -13200.358,E2 -13200.358} C_VEL
LIN {X 0,Y 364.864,Z 329.722,A -85,B 0,C 180,E1 -13201.757,E2 -13201.757} C_VEL
LIN {X 0,Y 365.791,Z 318.955,A -85,B 0,C 180,E1 -13202.851,E2 -13202.851} C_VEL
LIN {X 0,Y 366.659,Z 306.527,A -85,B 0,C 180,E1 -13203.842,E2 -13203.842} C_VEL
LIN {X 0,Y 364.416,Z 293.759,A -85,B 0,C 180,E1 -13204.743,E2 -13204.743} C_VEL
LIN {X 0,Y 361.351,Z 280.179,A -85,B 0,C 180,E1 -13205.474,E2 -13205.474} C_VEL
LIN {X 0,Y 360.773,Z 277.307,A -85,B 0,C 180,E1 -13205.624,E2 -13205.624} C_VEL
LIN {X 0,Y 361.045,Z 272.448,A -85,B 0,C 180,E1 -13209.49,E2 -13209.49} C_VEL
LIN {X 0,Y 361.284,Z 268.09,A -85,B 0,C 180,E1 -13213.035,E2 -13213.035} C_VEL
LIN {X 0,Y 361.52,Z 263.931,A -85,B 0,C 180,E1 -13216.51,E2 -13216.51} C_VEL
LIN {X 0,Y 361.734,Z 259.93,A -85,B 0,C 180,E1 -13219.93,E2 -13219.93} C_VEL
LIN {X 0,Y 361.817,Z 258.63,A -85,B 0,C 180,E1 -13221.061,E2 -13221.061} C_VEL
LIN {X 0,Y 362.103,Z 258.379,A -85,B 0,C 180,E1 -13223.313,E2 -13223.313} C_VEL
LIN {X 0,Y 362.273,Z 258.357,A -85,B 0,C 180,E1 -13227.777,E2 -13227.777} C_VEL
LIN {X 0,Y 362.419,Z 258.34,A -85,B 0,C 180,E1 -13230,E2 -13230} C_VEL
LIN {X 0,Y 362.273,Z 258.36,A -85,B 0,C 180,E1 -13232.224,E2 -13232.224} C_VEL
LIN {X 0,Y 362.161,Z 258.373,A -85,B 0,C 180,E1 -13236.686,E2 -13236.686} C_VEL
LIN {X 0,Y 362.065,Z 258.384,A -85,B 0,C 180,E1 -13238.933,E2 -13238.933} C_VEL
LIN {X 0,Y 361.957,Z 258.401,A -85,B 0,C 180,E1 -13242.332,E2 -13242.332} C_VEL
LIN {X 0,Y 361.953,Z 258.398,A -85,B 0,C 180,E1 -13244.621,E2 -13244.621} C_VEL
LIN {X 0,Y 361.95,Z 258.401,A -85,B 0,C 180,E1 -13248.1,E2 -13248.1} C_VEL
LIN {X 0,Y 361.892,Z 258.407,A -85,B 0,C 180,E1 -13251.653,E2 -13251.653} C_VEL
LIN {X 0,Y 361.919,Z 258.402,A -85,B 0,C 180,E1 -13255.29,E2 -13255.29} C_VEL
LIN {X 0,Y 361.912,Z 258.406,A -85,B 0,C 180,E1 -13257.778,E2 -13257.778} C_VEL
LIN {X 0,Y 361.849,Z 258.414,A -85,B 0,C 180,E1 -13261.628,E2 -13261.628} C_VEL
LIN {X 0,Y 361.838,Z 258.411,A -85,B 0,C 180,E1 -13264.556,E2 -13264.556} C_VEL
LIN {X 0,Y 361.179,Z 258.497,A -85,B 0,C 180,E1 -13265.486,E2 -13265.486} C_VEL
LIN {X 0,Y 358.355,Z 258.854,A -85,B 0,C 180,E1 -13266.998,E2 -13266.998} C_VEL
LIN {X 0,Y 355.951,Z 259.155,A -85,B 0,C 180,E1 -13268.221,E2 -13268.221} C_VEL
LIN {X 0,Y 354.904,Z 259.281,A -85,B 0,C 180,E1 -13269.167,E2 -13269.167} C_VEL
LIN {X 0,Y 354.811,Z 259.29,A -85,B 0,C 180,E1 -13269.488,E2 -13269.488} C_VEL
LIN {X 0,Y 354.832,Z 259.284,A -85,B 0,C 180,E1 -13272.877,E2 -13272.877} C_VEL
LIN {X 0,Y 354.856,Z 259.281,A -85,B 0,C 180,E1 -13276.12,E2 -13276.12} C_VEL
LIN {X 0,Y 354.846,Z 259.286,A -85,B 0,C 180,E1 -13279.189,E2 -13279.189} C_VEL
LIN {X 0,Y 354.8,Z 259.288,A -85,B 0,C 180,E1 -13282.403,E2 -13282.403} C_VEL
LIN {X 0,Y 354.803,Z 259.291,A -85,B 0,C 180,E1 -13284.942,E2 -13284.942} C_VEL
LIN {X 0,Y 354.784,Z 259.29,A -85,B 0,C 180,E1 -13288.406,E2 -13288.406} C_VEL
LIN {X 0,Y 354.845,Z 259.282,A -85,B 0,C 180,E1 -13291.62,E2 -13291.62} C_VEL
LIN {X 0,Y 354.891,Z 259.276,A -85,B 0,C 180,E1 -13294.174,E2 -13294.174} C_VEL
LIN {X 0,Y 354.826,Z 259.284,A -85,B 0,C 180,E1 -13297.895,E2 -13297.895} C_VEL
LIN {X 0,Y 354.915,Z 259.273,A -85,B 0,C 180,E1 -13301.893,E2 -13301.893} C_VEL
LIN {X 0,Y 354.935,Z 259.271,A -85,B 0,C 180,E1 -13305.983,E2 -13305.983} C_VEL
LIN {X 0,Y 354.972,Z 259.266,A -85,B 0,C 180,E1 -13309.737,E2 -13309.737} C_VEL
LIN {X 0,Y 355.12,Z 259.248,A -85,B 0,C 180,E1 -13313.182,E2 -13313.182} C_VEL
LIN {X 0,Y 355.24,Z 259.234,A -85,B 0,C 180,E1 -13317.734,E2 -13317.734} C_VEL
LIN {X 0,Y 355.392,Z 259.217,A -85,B 0,C 180,E1 -13320.001,E2 -13320.001} C_VEL
LIN {X 0,Y 355.241,Z 259.237,A -85,B 0,C 180,E1 -13322.269,E2 -13322.269} C_VEL
LIN {X 0,Y 355.133,Z 259.246,A -85,B 0,C 180,E1 -13326.821,E2 -13326.821} C_VEL
LIN {X 0,Y 355.013,Z 259.261,A -85,B 0,C 180,E1 -13329.114,E2 -13329.114} C_VEL
LIN {X 0,Y 354.922,Z 259.273,A -85,B 0,C 180,E1 -13332.582,E2 -13332.582} C_VEL
LIN {X 0,Y 354.887,Z 259.28,A -85,B 0,C 180,E1 -13336.097,E2 -13336.097} C_VEL
LIN {X 0,Y 354.899,Z 259.276,A -85,B 0,C 180,E1 -13338.473,E2 -13338.473} C_VEL
LIN {X 0,Y 354.833,Z 259.285,A -85,B 0,C 180,E1 -13342.107,E2 -13342.107} C_VEL
LIN {X 0,Y 354.897,Z 259.278,A -85,B 0,C 180,E1 -13345.829,E2 -13345.829} C_VEL
LIN {X 0,Y 354.817,Z 259.289,A -85,B 0,C 180,E1 -13349.683,E2 -13349.683} C_VEL
LIN {X 0,Y 354.806,Z 259.289,A -85,B 0,C 180,E1 -13353.703,E2 -13353.703} C_VEL
LIN {X 0,Y 354.801,Z 259.287,A -85,B 0,C 180,E1 -13356.46,E2 -13356.46} C_VEL
LIN {X 0,Y 354.825,Z 259.288,A -85,B 0,C 180,E1 -13359.425,E2 -13359.425} C_VEL
LIN {X 0,Y 354.789,Z 259.292,A -85,B 0,C 180,E1 -13362.868,E2 -13362.868} C_VEL
LIN {X 0,Y 354.769,Z 259.295,A -85,B 0,C 180,E1 -13366.105,E2 -13366.105} C_VEL
LIN {X 0,Y 354.843,Z 259.311,A -85,B 0,C 180,E1 -13367.671,E2 -13367.671} C_VEL
LIN {X 0,Y 355.616,Z 263.739,A -85,B 0,C 180,E1 -13370.772,E2 -13370.772} C_VEL
LIN {X 0,Y 356.105,Z 268.133,A -85,B 0,C 180,E1 -13373.696,E2 -13373.696} C_VEL
LIN {X 0,Y 356.046,Z 271.768,A -85,B 0,C 180,E1 -13376.002,E2 -13376.002} C_VEL
LIN {X 0,Y 355.312,Z 277.888,A -85,B 0,C 180,E1 -13379.71,E2 -13379.71} C_VEL
LIN {X 0,Y 354.663,Z 285.434,A -85,B 0,C 180,E1 -13384.154,E2 -13384.154} C_VEL
LIN {X 0,Y 354.217,Z 291.874,A -85,B 0,C 180,E1 -13387.854,E2 -13387.854} C_VEL
LIN {X 0,Y 353.98,Z 295.797,A -85,B 0,C 180,E1 -13390.067,E2 -13390.067} C_VEL
LIN {X 0,Y 356.364,Z 309.281,A -85,B 0,C 180,E1 -13390.698,E2 -13390.698} C_VEL
LIN {X 0,Y 358.228,Z 322.304,A -85,B 0,C 180,E1 -13391.528,E2 -13391.528} C_VEL
LIN {X 0,Y 359.102,Z 332.649,A -85,B 0,C 180,E1 -13392.341,E2 -13392.341} C_VEL
LIN {X 0,Y 357.941,Z 344.883,A -85,B 0,C 180,E1 -13393.459,E2 -13393.459} C_VEL
LIN {X 0,Y 356.842,Z 355.676,A -85,B 0,C 180,E1 -13394.725,E2 -13394.725} C_VEL
LIN {X 0,Y 355.841,Z 366.344,A -85,B 0,C 180,E1 -13396.29,E2 -13396.29} C_VEL
LIN {X 0,Y 355.052,Z 374.197,A -85,B 0,C 180,E1 -13397.714,E2 -13397.714} C_VEL
LIN {X 0,Y 354.313,Z 381.863,A -85,B 0,C 180,E1 -13399.428,E2 -13399.428} C_VEL
LIN {X 0,Y 353.729,Z 388.94,A -85,B 0,C 180,E1 -13401.43,E2 -13401.43} C_VEL
LIN {X 0,Y 353.419,Z 393.623,A -85,B 0,C 180,E1 -13403.147,E2 -13403.147} C_VEL
LIN {X 0,Y 353.263,Z 397.177,A -85,B 0,C 180,E1 -13404.864,E2 -13404.864} C_VEL
LIN {X 0,Y 353.224,Z 399.704,A -85,B 0,C 180,E1 -13406.578,E2 -13406.578} C_VEL
LIN {X 0,Y 353.176,Z 400.87,A -85,B 0,C 180,E1 -13407.719,E2 -13407.719} C_VEL
LIN {X 0,Y 353.219,Z 401.589,A -85,B 0,C 180,E1 -13408.86,E2 -13408.86} C_VEL
